LIN {X 0,Y 580.04,Z 560.279,A -85,B 0,C 180,E1 -1982.083,E2 -1982.083} C_VEL
LIN {X 0,Y 580.123,Z 557.073,A -85,B 0,C 180,E1 -1983.473,E2 -1983.473} C_VEL
LIN {X 0,Y 580.108,Z 553.521,A -85,B 0,C 180,E1 -1984.517,E2 -1984.517} C_VEL
LIN {X 0,Y 580.137,Z 548.87,A -85,B 0,C 180,E1 -1985.562,E2 -1985.562} C_VEL
LIN {X 0,Y 580.13,Z 542.972,A -85,B 0,C 180,E1 -1986.611,E2 -1986.611} C_VEL
LIN {X 0,Y 580.221,Z 535.668,A -85,B 0,C 180,E1 -1987.657,E2 -1987.657} C_VEL
LIN {X 0,Y 580.259,Z 526.563,A -85,B 0,C 180,E1 -1988.708,E2 -1988.708} C_VEL
LIN {X 0,Y 580.369,Z 515.986,A -85,B 0,C 180,E1 -1989.673,E2 -1989.673} C_VEL
LIN {X 0,Y 580.453,Z 506.507,A -85,B 0,C 180,E1 -1990.376,E2 -1990.376} C_VEL
LIN {X 0,Y 580.558,Z 496.346,A -85,B 0,C 180,E1 -1990.992,E2 -1990.992} C_VEL
LIN {X 0,Y 580.6,Z 486.208,A -85,B 0,C 180,E1 -1991.486,E2 -1991.486} C_VEL
LIN {X 0,Y 580.71,Z 474.792,A -85,B 0,C 180,E1 -1991.917,E2 -1991.917} C_VEL
LIN {X 0,Y 580.801,Z 461.468,A -85,B 0,C 180,E1 -1992.27,E2 -1992.27} C_VEL
LIN {X 0,Y 580.831,Z 443.197,A -85,B 0,C 180,E1 -1992.535,E2 -1992.535} C_VEL
LIN {X 0,Y 580.93,Z 408.349,A -85,B 0,C 180,E1 -1992.966,E2 -1992.966} C_VEL
LIN {X 0,Y 580.085,Z 398.577,A -85,B 0,C 180,E1 -1993.118,E2 -1993.118} C_VEL
LIN {X 0,Y 578.705,Z 392.854,A -85,B 0,C 180,E1 -1993.21,E2 -1993.21} C_VEL
LIN {X 0,Y 574.137,Z 379.962,A -85,B 0,C 180,E1 -1993.479,E2 -1993.479} C_VEL
LIN {X 0,Y 573.484,Z 378.185,A -85,B 0,C 180,E1 -1993.53,E2 -1993.53} C_VEL
LIN {X 0,Y 573.292,Z 377.197,A -85,B 0,C 180,E1 -1993.65,E2 -1993.65} C_VEL
LIN {X 0,Y 573.25,Z 377.078,A -85,B 0,C 180,E1 -1996.378,E2 -1996.378} C_VEL
LIN {X 0,Y 573.27,Z 377.074,A -85,B 0,C 180,E1 -1999.33,E2 -1999.33} C_VEL
LIN {X 0,Y 573.237,Z 377.078,A -85,B 0,C 180,E1 -2002.338,E2 -2002.338} C_VEL
LIN {X 0,Y 573.248,Z 377.074,A -85,B 0,C 180,E1 -2005.411,E2 -2005.411} C_VEL
LIN {X 0,Y 573.232,Z 377.081,A -85,B 0,C 180,E1 -2008.565,E2 -2008.565} C_VEL
LIN {X 0,Y 573.227,Z 377.082,A -85,B 0,C 180,E1 -2010.993,E2 -2010.993} C_VEL
LIN {X 0,Y 573.244,Z 377.072,A -85,B 0,C 180,E1 -2013.521,E2 -2013.521} C_VEL
LIN {X 0,Y 573.197,Z 377.081,A -85,B 0,C 180,E1 -2016.053,E2 -2016.053} C_VEL
LIN {X 0,Y 573.242,Z 377.083,A -85,B 0,C 180,E1 -2018.702,E2 -2018.702} C_VEL
LIN {X 0,Y 573.23,Z 377.075,A -85,B 0,C 180,E1 -2021.593,E2 -2021.593} C_VEL
LIN {X 0,Y 573.22,Z 377.082,A -85,B 0,C 180,E1 -2024.335,E2 -2024.335} C_VEL
LIN {X 0,Y 573.236,Z 377.075,A -85,B 0,C 180,E1 -2027.359,E2 -2027.359} C_VEL
LIN {X 0,Y 573.239,Z 377.082,A -85,B 0,C 180,E1 -2030.392,E2 -2030.392} C_VEL
LIN {X 0,Y 573.233,Z 377.078,A -85,B 0,C 180,E1 -2033.076,E2 -2033.076} C_VEL
LIN {X 0,Y 573.265,Z 377.071,A -85,B 0,C 180,E1 -2035.671,E2 -2035.671} C_VEL
LIN {X 0,Y 573.238,Z 377.078,A -85,B 0,C 180,E1 -2038.184,E2 -2038.184} C_VEL
LIN {X 0,Y 573.258,Z 377.081,A -85,B 0,C 180,E1 -2040.634,E2 -2040.634} C_VEL
LIN {X 0,Y 573.297,Z 377.287,A -85,B 0,C 180,E1 -2043.388,E2 -2043.388} C_VEL
LIN {X 0,Y 574.525,Z 382.647,A -85,B 0,C 180,E1 -2044.067,E2 -2044.067} C_VEL
LIN {X 0,Y 574.55,Z 397.786,A -85,B 0,C 180,E1 -2045.809,E2 -2045.809} C_VEL
LIN {X 0,Y 574.254,Z 421.464,A -85,B 0,C 180,E1 -2048.586,E2 -2048.586} C_VEL
LIN {X 0,Y 573.914,Z 446.146,A -85,B 0,C 180,E1 -2051.434,E2 -2051.434} C_VEL
LIN {X 0,Y 573.616,Z 471.912,A -85,B 0,C 180,E1 -2054.363,E2 -2054.363} C_VEL
LIN {X 0,Y 573.514,Z 488.192,A -85,B 0,C 180,E1 -2056.175,E2 -2056.175} C_VEL
LIN {X 0,Y 574.082,Z 493.73,A -85,B 0,C 180,E1 -2056.279,E2 -2056.279} C_VEL
LIN {X 0,Y 573.886,Z 597.916,A -85,B 0,C 180,E1 -2057.602,E2 -2057.602} C_VEL
LIN {X 0,Y 573.831,Z 610.341,A -85,B 0,C 180,E1 -2057.893,E2 -2057.893} C_VEL
LIN {X 0,Y 573.705,Z 622.21,A -85,B 0,C 180,E1 -2058.294,E2 -2058.294} C_VEL
LIN {X 0,Y 573.588,Z 634.849,A -85,B 0,C 180,E1 -2058.876,E2 -2058.876} C_VEL
LIN {X 0,Y 573.445,Z 646.523,A -85,B 0,C 180,E1 -2059.585,E2 -2059.585} C_VEL
LIN {X 0,Y 573.35,Z 655.955,A -85,B 0,C 180,E1 -2060.297,E2 -2060.297} C_VEL
LIN {X 0,Y 573.262,Z 663.842,A -85,B 0,C 180,E1 -2061.007,E2 -2061.007} C_VEL
LIN {X 0,Y 573.178,Z 672.073,A -85,B 0,C 180,E1 -2061.894,E2 -2061.894} C_VEL
LIN {X 0,Y 573.105,Z 680.149,A -85,B 0,C 180,E1 -2062.956,E2 -2062.956} C_VEL
LIN {X 0,Y 573.093,Z 686.626,A -85,B 0,C 180,E1 -2064.017,E2 -2064.017} C_VEL
LIN {X 0,Y 572.962,Z 691.755,A -85,B 0,C 180,E1 -2065.074,E2 -2065.074} C_VEL
LIN {X 0,Y 573.014,Z 695.735,A -85,B 0,C 180,E1 -2066.132,E2 -2066.132} C_VEL
LIN {X 0,Y 572.959,Z 698.688,A -85,B 0,C 180,E1 -2067.188,E2 -2067.188} C_VEL
LIN {X 0,Y 572.939,Z 700.137,A -85,B 0,C 180,E1 -2067.891,E2 -2067.891} C_VEL
LIN {X 0,Y 572.941,Z 701.756,A -85,B 0,C 180,E1 -2069.297,E2 -2069.297} C_VEL
LIN {X 0,Y 572.939,Z 701.996,A -85,B 0,C 180,E1 -2070,E2 -2070} C_VEL
LIN {X 0,Y 572.947,Z 701.229,A -85,B 0,C 180,E1 -2071.406,E2 -2071.406} C_VEL
LIN {X 0,Y 572.939,Z 700.28,A -85,B 0,C 180,E1 -2072.109,E2 -2072.109} C_VEL
LIN {X 0,Y 572.959,Z 698.879,A -85,B 0,C 180,E1 -2072.812,E2 -2072.812} C_VEL
LIN {X 0,Y 573.015,Z 696.005,A -85,B 0,C 180,E1 -2073.868,E2 -2073.868} C_VEL
LIN {X 0,Y 572.962,Z 692.116,A -85,B 0,C 180,E1 -2074.926,E2 -2074.926} C_VEL
LIN {X 0,Y 573.071,Z 687.095,A -85,B 0,C 180,E1 -2075.984,E2 -2075.984} C_VEL
LIN {X 0,Y 573.114,Z 679.539,A -85,B 0,C 180,E1 -2077.221,E2 -2077.221} C_VEL
LIN {X 0,Y 573.169,Z 672.832,A -85,B 0,C 180,E1 -2078.106,E2 -2078.106} C_VEL
LIN {X 0,Y 573.251,Z 664.745,A -85,B 0,C 180,E1 -2078.993,E2 -2078.993} C_VEL
LIN {X 0,Y 573.342,Z 654.904,A -85,B 0,C 180,E1 -2079.882,E2 -2079.882} C_VEL
LIN {X 0,Y 573.516,Z 643.899,A -85,B 0,C 180,E1 -2080.681,E2 -2080.681} C_VEL
LIN {X 0,Y 573.636,Z 631.59,A -85,B 0,C 180,E1 -2081.377,E2 -2081.377} C_VEL
LIN {X 0,Y 573.701,Z 620.22,A -85,B 0,C 180,E1 -2081.872,E2 -2081.872} C_VEL
LIN {X 0,Y 573.802,Z 608.017,A -85,B 0,C 180,E1 -2082.265,E2 -2082.265} C_VEL
LIN {X 0,Y 573.922,Z 595.156,A -85,B 0,C 180,E1 -2082.532,E2 -2082.532} C_VEL
LIN {X 0,Y 573.944,Z 491.455,A -85,B 0,C 180,E1 -2083.843,E2 -2083.843} C_VEL
LIN {X 0,Y 573.528,Z 488.15,A -85,B 0,C 180,E1 -2083.915,E2 -2083.915} C_VEL
LIN {X 0,Y 573.733,Z 461.428,A -85,B 0,C 180,E1 -2086.914,E2 -2086.914} C_VEL
LIN {X 0,Y 574.055,Z 435.714,A -85,B 0,C 180,E1 -2089.853,E2 -2089.853} C_VEL
LIN {X 0,Y 574.423,Z 409.87,A -85,B 0,C 180,E1 -2092.859,E2 -2092.859} C_VEL
LIN {X 0,Y 574.656,Z 388.489,A -85,B 0,C 180,E1 -2095.344,E2 -2095.344} C_VEL
LIN {X 0,Y 574.626,Z 383.426,A -85,B 0,C 180,E1 -2095.928,E2 -2095.928} C_VEL
LIN {X 0,Y 573.246,Z 377.157,A -85,B 0,C 180,E1 -2096.74,E2 -2096.74} C_VEL
LIN {X 0,Y 573.226,Z 377.079,A -85,B 0,C 180,E1 -2099.484,E2 -2099.484} C_VEL
LIN {X 0,Y 573.24,Z 377.077,A -85,B 0,C 180,E1 -2102.226,E2 -2102.226} C_VEL
LIN {X 0,Y 573.225,Z 377.077,A -85,B 0,C 180,E1 -2104.769,E2 -2104.769} C_VEL
LIN {X 0,Y 573.223,Z 377.084,A -85,B 0,C 180,E1 -2107.809,E2 -2107.809} C_VEL
LIN {X 0,Y 573.249,Z 377.071,A -85,B 0,C 180,E1 -2110.525,E2 -2110.525} C_VEL
LIN {X 0,Y 573.207,Z 377.086,A -85,B 0,C 180,E1 -2113.665,E2 -2113.665} C_VEL
LIN {X 0,Y 573.204,Z 377.078,A -85,B 0,C 180,E1 -2116.637,E2 -2116.637} C_VEL
LIN {X 0,Y 573.249,Z 377.08,A -85,B 0,C 180,E1 -2119.475,E2 -2119.475} C_VEL
LIN {X 0,Y 573.221,Z 377.078,A -85,B 0,C 180,E1 -2122.191,E2 -2122.191} C_VEL
LIN {X 0,Y 573.222,Z 377.079,A -85,B 0,C 180,E1 -2125.231,E2 -2125.231} C_VEL
LIN {X 0,Y 573.252,Z 377.082,A -85,B 0,C 180,E1 -2127.773,E2 -2127.773} C_VEL
LIN {X 0,Y 573.225,Z 377.075,A -85,B 0,C 180,E1 -2130.632,E2 -2130.632} C_VEL
LIN {X 0,Y 573.201,Z 377.086,A -85,B 0,C 180,E1 -2133.516,E2 -2133.516} C_VEL
LIN {X 0,Y 573.219,Z 377.078,A -85,B 0,C 180,E1 -2136.134,E2 -2136.134} C_VEL
LIN {X 0,Y 573.234,Z 377.077,A -85,B 0,C 180,E1 -2139.173,E2 -2139.173} C_VEL
LIN {X 0,Y 573.202,Z 377.083,A -85,B 0,C 180,E1 -2141.41,E2 -2141.41} C_VEL
LIN {X 0,Y 573.211,Z 377.079,A -85,B 0,C 180,E1 -2144.351,E2 -2144.351} C_VEL
LIN {X 0,Y 573.214,Z 377.077,A -85,B 0,C 180,E1 -2146.529,E2 -2146.529} C_VEL
LIN {X 0,Y 573.242,Z 377.075,A -85,B 0,C 180,E1 -2149.403,E2 -2149.403} C_VEL
LIN {X 0,Y 573.223,Z 377.078,A -85,B 0,C 180,E1 -2152.249,E2 -2152.249} C_VEL
LIN {X 0,Y 573.281,Z 377.067,A -85,B 0,C 180,E1 -2155.077,E2 -2155.077} C_VEL
LIN {X 0,Y 573.309,Z 377.073,A -85,B 0,C 180,E1 -2157.892,E2 -2157.892} C_VEL
LIN {X 0,Y 573.32,Z 377.069,A -85,B 0,C 180,E1 -2160,E2 -2160} C_VEL
LIN {X 0,Y 573.273,Z 377.066,A -85,B 0,C 180,E1 -2162.811,E2 -2162.811} C_VEL
LIN {X 0,Y 573.27,Z 377.077,A -85,B 0,C 180,E1 -2165.628,E2 -2165.628} C_VEL
LIN {X 0,Y 573.238,Z 377.073,A -85,B 0,C 180,E1 -2168.46,E2 -2168.46} C_VEL
LIN {X 0,Y 573.24,Z 377.075,A -85,B 0,C 180,E1 -2171.313,E2 -2171.313} C_VEL
LIN {X 0,Y 573.246,Z 377.074,A -85,B 0,C 180,E1 -2174.408,E2 -2174.408} C_VEL
LIN {X 0,Y 573.18,Z 377.079,A -85,B 0,C 180,E1 -2177.114,E2 -2177.114} C_VEL
LIN {X 0,Y 573.204,Z 377.084,A -85,B 0,C 180,E1 -2180.078,E2 -2180.078} C_VEL
LIN {X 0,Y 573.218,Z 377.077,A -85,B 0,C 180,E1 -2182.339,E2 -2182.339} C_VEL
LIN {X 0,Y 573.209,Z 377.081,A -85,B 0,C 180,E1 -2185.412,E2 -2185.412} C_VEL
LIN {X 0,Y 573.195,Z 377.084,A -85,B 0,C 180,E1 -2188.017,E2 -2188.017} C_VEL
LIN {X 0,Y 573.22,Z 377.076,A -85,B 0,C 180,E1 -2190.88,E2 -2190.88} C_VEL
LIN {X 0,Y 573.245,Z 377.078,A -85,B 0,C 180,E1 -2193.521,E2 -2193.521} C_VEL
LIN {X 0,Y 573.184,Z 377.088,A -85,B 0,C 180,E1 -2196.054,E2 -2196.054} C_VEL
LIN {X 0,Y 573.215,Z 377.076,A -85,B 0,C 180,E1 -2198.704,E2 -2198.704} C_VEL
LIN {X 0,Y 573.187,Z 377.08,A -85,B 0,C 180,E1 -2201.587,E2 -2201.587} C_VEL
LIN {X 0,Y 573.207,Z 377.081,A -85,B 0,C 180,E1 -2204.336,E2 -2204.336} C_VEL
LIN {X 0,Y 573.195,Z 377.079,A -85,B 0,C 180,E1 -2206.636,E2 -2206.636} C_VEL
LIN {X 0,Y 573.202,Z 377.077,A -85,B 0,C 180,E1 -2209.48,E2 -2209.48} C_VEL
LIN {X 0,Y 573.209,Z 377.084,A -85,B 0,C 180,E1 -2212.19,E2 -2212.19} C_VEL
LIN {X 0,Y 573.211,Z 377.079,A -85,B 0,C 180,E1 -2215.233,E2 -2215.233} C_VEL
LIN {X 0,Y 573.223,Z 377.085,A -85,B 0,C 180,E1 -2217.777,E2 -2217.777} C_VEL
LIN {X 0,Y 573.219,Z 377.081,A -85,B 0,C 180,E1 -2220.631,E2 -2220.631} C_VEL
LIN {X 0,Y 573.226,Z 377.225,A -85,B 0,C 180,E1 -2222.751,E2 -2222.751} C_VEL
LIN {X 0,Y 574.782,Z 383.948,A -85,B 0,C 180,E1 -2223.589,E2 -2223.589} C_VEL
LIN {X 0,Y 574.627,Z 405.704,A -85,B 0,C 180,E1 -2226.004,E2 -2226.004} C_VEL
LIN {X 0,Y 574.261,Z 431.045,A -85,B 0,C 180,E1 -2228.85,E2 -2228.85} C_VEL
LIN {X 0,Y 573.894,Z 457.816,A -85,B 0,C 180,E1 -2231.803,E2 -2231.803} C_VEL
LIN {X 0,Y 573.643,Z 483.031,A -85,B 0,C 180,E1 -2234.545,E2 -2234.545} C_VEL
LIN {X 0,Y 573.519,Z 497.889,A -85,B 0,C 180,E1 -2236.13,E2 -2236.13} C_VEL
LIN {X 0,Y 574.08,Z 503.704,A -85,B 0,C 180,E1 -2236.234,E2 -2236.234} C_VEL
LIN {X 0,Y 573.882,Z 607.937,A -85,B 0,C 180,E1 -2237.557,E2 -2237.557} C_VEL
LIN {X 0,Y 573.785,Z 621.213,A -85,B 0,C 180,E1 -2237.869,E2 -2237.869} C_VEL
LIN {X 0,Y 573.702,Z 634.147,A -85,B 0,C 180,E1 -2238.325,E2 -2238.325} C_VEL
LIN {X 0,Y 573.591,Z 645.717,A -85,B 0,C 180,E1 -2238.878,E2 -2238.878} C_VEL
LIN {X 0,Y 573.438,Z 657.2,A -85,B 0,C 180,E1 -2239.585,E2 -2239.585} C_VEL
LIN {X 0,Y 573.331,Z 667.598,A -85,B 0,C 180,E1 -2240.385,E2 -2240.385} C_VEL
LIN {X 0,Y 573.241,Z 676.111,A -85,B 0,C 180,E1 -2241.184,E2 -2241.184} C_VEL
LIN {X 0,Y 573.161,Z 683.959,A -85,B 0,C 180,E1 -2242.071,E2 -2242.071} C_VEL
LIN {X 0,Y 573.073,Z 691.953,A -85,B 0,C 180,E1 -2243.185,E2 -2243.185} C_VEL
LIN {X 0,Y 573.07,Z 698.679,A -85,B 0,C 180,E1 -2244.37,E2 -2244.37} C_VEL
LIN {X 0,Y 573.028,Z 703.371,A -85,B 0,C 180,E1 -2245.427,E2 -2245.427} C_VEL
LIN {X 0,Y 573.022,Z 706.957,A -85,B 0,C 180,E1 -2246.484,E2 -2246.484} C_VEL
LIN {X 0,Y 572.959,Z 708.808,A -85,B 0,C 180,E1 -2247.188,E2 -2247.188} C_VEL
LIN {X 0,Y 572.939,Z 710.198,A -85,B 0,C 180,E1 -2247.891,E2 -2247.891} C_VEL
LIN {X 0,Y 572.94,Z 711.785,A -85,B 0,C 180,E1 -2249.297,E2 -2249.297} C_VEL
LIN {X 0,Y 572.938,Z 712,A -85,B 0,C 180,E1 -2250,E2 -2250} C_VEL
LIN {X 0,Y 572.946,Z 711.186,A -85,B 0,C 180,E1 -2251.406,E2 -2251.406} C_VEL
LIN {X 0,Y 572.939,Z 710.2,A -85,B 0,C 180,E1 -2252.109,E2 -2252.109} C_VEL
LIN {X 0,Y 572.959,Z 708.81,A -85,B 0,C 180,E1 -2252.812,E2 -2252.812} C_VEL
LIN {X 0,Y 573.015,Z 705.896,A -85,B 0,C 180,E1 -2253.868,E2 -2253.868} C_VEL
LIN {X 0,Y 572.963,Z 701.949,A -85,B 0,C 180,E1 -2254.926,E2 -2254.926} C_VEL
LIN {X 0,Y 573.064,Z 695.877,A -85,B 0,C 180,E1 -2256.16,E2 -2256.16} C_VEL
LIN {X 0,Y 573.119,Z 689.238,A -85,B 0,C 180,E1 -2257.221,E2 -2257.221} C_VEL
LIN {X 0,Y 573.201,Z 680.991,A -85,B 0,C 180,E1 -2258.283,E2 -2258.283} C_VEL
LIN {X 0,Y 573.287,Z 672.539,A -85,B 0,C 180,E1 -2259.17,E2 -2259.17} C_VEL
LIN {X 0,Y 573.425,Z 662.098,A -85,B 0,C 180,E1 -2260.058,E2 -2260.058} C_VEL
LIN {X 0,Y 573.534,Z 651.772,A -85,B 0,C 180,E1 -2260.769,E2 -2260.769} C_VEL
LIN {X 0,Y 573.628,Z 640.588,A -85,B 0,C 180,E1 -2261.385,E2 -2261.385} C_VEL
LIN {X 0,Y 573.719,Z 628.768,A -85,B 0,C 180,E1 -2261.885,E2 -2261.885} C_VEL
LIN {X 0,Y 573.822,Z 615.349,A -85,B 0,C 180,E1 -2262.287,E2 -2262.287} C_VEL
LIN {X 0,Y 573.951,Z 602.085,A -85,B 0,C 180,E1 -2262.531,E2 -2262.531} C_VEL
LIN {X 0,Y 573.89,Z 500.813,A -85,B 0,C 180,E1 -2263.807,E2 -2263.807} C_VEL
LIN {X 0,Y 573.519,Z 497.888,A -85,B 0,C 180,E1 -2263.87,E2 -2263.87} C_VEL
LIN {X 0,Y 573.782,Z 472.947,A -85,B 0,C 180,E1 -2266.546,E2 -2266.546} C_VEL
LIN {X 0,Y 574.04,Z 446.069,A -85,B 0,C 180,E1 -2269.487,E2 -2269.487} C_VEL
LIN {X 0,Y 574.394,Z 420.835,A -85,B 0,C 180,E1 -2272.29,E2 -2272.29} C_VEL
LIN {X 0,Y 574.659,Z 399.163,A -85,B 0,C 180,E1 -2274.721,E2 -2274.721} C_VEL
LIN {X 0,Y 574.682,Z 383.397,A -85,B 0,C 180,E1 -2276.416,E2 -2276.416} C_VEL
LIN {X 0,Y 573.222,Z 377.203,A -85,B 0,C 180,E1 -2277.175,E2 -2277.175} C_VEL
LIN {X 0,Y 573.218,Z 377.086,A -85,B 0,C 180,E1 -2280.178,E2 -2280.178} C_VEL
LIN {X 0,Y 573.217,Z 377.079,A -85,B 0,C 180,E1 -2282.647,E2 -2282.647} C_VEL
LIN {X 0,Y 573.18,Z 377.084,A -85,B 0,C 180,E1 -2285.19,E2 -2285.19} C_VEL
LIN {X 0,Y 573.211,Z 377.087,A -85,B 0,C 180,E1 -2287.81,E2 -2287.81} C_VEL
LIN {X 0,Y 573.201,Z 377.08,A -85,B 0,C 180,E1 -2290.529,E2 -2290.529} C_VEL
LIN {X 0,Y 573.196,Z 377.084,A -85,B 0,C 180,E1 -2293.363,E2 -2293.363} C_VEL
LIN {X 0,Y 573.206,Z 377.08,A -85,B 0,C 180,E1 -2296.335,E2 -2296.335} C_VEL
LIN {X 0,Y 573.204,Z 377.079,A -85,B 0,C 180,E1 -2298.54,E2 -2298.54} C_VEL
LIN {X 0,Y 573.233,Z 377.08,A -85,B 0,C 180,E1 -2301.297,E2 -2301.297} C_VEL
LIN {X 0,Y 573.188,Z 377.085,A -85,B 0,C 180,E1 -2304.022,E2 -2304.022} C_VEL
LIN {X 0,Y 573.242,Z 377.075,A -85,B 0,C 180,E1 -2306.516,E2 -2306.516} C_VEL
LIN {X 0,Y 573.228,Z 377.08,A -85,B 0,C 180,E1 -2309.119,E2 -2309.119} C_VEL
LIN {X 0,Y 573.228,Z 377.085,A -85,B 0,C 180,E1 -2311.435,E2 -2311.435} C_VEL
LIN {X 0,Y 573.24,Z 377.075,A -85,B 0,C 180,E1 -2314.589,E2 -2314.589} C_VEL
LIN {X 0,Y 573.235,Z 377.081,A -85,B 0,C 180,E1 -2317.662,E2 -2317.662} C_VEL
LIN {X 0,Y 573.269,Z 377.073,A -85,B 0,C 180,E1 -2320.67,E2 -2320.67} C_VEL
LIN {X 0,Y 573.251,Z 377.08,A -85,B 0,C 180,E1 -2323.622,E2 -2323.622} C_VEL
LIN {X 0,Y 573.299,Z 377.197,A -85,B 0,C 180,E1 -2326.441,E2 -2326.441} C_VEL
LIN {X 0,Y 573.526,Z 378.312,A -85,B 0,C 180,E1 -2326.567,E2 -2326.567} C_VEL
LIN {X 0,Y 574.033,Z 380.55,A -85,B 0,C 180,E1 -2326.616,E2 -2326.616} C_VEL
LIN {X 0,Y 573.912,Z 457.586,A -85,B 0,C 180,E1 -2327.603,E2 -2327.603} C_VEL
LIN {X 0,Y 573.807,Z 468.697,A -85,B 0,C 180,E1 -2327.848,E2 -2327.848} C_VEL
LIN {X 0,Y 573.718,Z 481.135,A -85,B 0,C 180,E1 -2328.249,E2 -2328.249} C_VEL
LIN {X 0,Y 573.622,Z 493.628,A -85,B 0,C 180,E1 -2328.813,E2 -2328.813} C_VEL
LIN {X 0,Y 573.488,Z 503.829,A -85,B 0,C 180,E1 -2329.408,E2 -2329.408} C_VEL
LIN {X 0,Y 573.343,Z 513.737,A -85,B 0,C 180,E1 -2330.118,E2 -2330.118} C_VEL
LIN {X 0,Y 573.287,Z 521.975,A -85,B 0,C 180,E1 -2330.83,E2 -2330.83} C_VEL
LIN {X 0,Y 573.187,Z 530.527,A -85,B 0,C 180,E1 -2331.717,E2 -2331.717} C_VEL
LIN {X 0,Y 573.114,Z 537.611,A -85,B 0,C 180,E1 -2332.602,E2 -2332.602} C_VEL
LIN {X 0,Y 573.049,Z 544.597,A -85,B 0,C 180,E1 -2333.663,E2 -2333.663} C_VEL
LIN {X 0,Y 573.009,Z 550.176,A -85,B 0,C 180,E1 -2334.722,E2 -2334.722} C_VEL
LIN {X 0,Y 573.031,Z 554.536,A -85,B 0,C 180,E1 -2335.78,E2 -2335.78} C_VEL
LIN {X 0,Y 572.959,Z 558.66,A -85,B 0,C 180,E1 -2337.188,E2 -2337.188} C_VEL
LIN {X 0,Y 572.939,Z 560.134,A -85,B 0,C 180,E1 -2337.891,E2 -2337.891} C_VEL
LIN {X 0,Y 572.941,Z 561.735,A -85,B 0,C 180,E1 -2339.297,E2 -2339.297} C_VEL
LIN {X 0,Y 572.939,Z 561.996,A -85,B 0,C 180,E1 -2340,E2 -2340} C_VEL
LIN {X 0,Y 572.947,Z 561.225,A -85,B 0,C 180,E1 -2341.406,E2 -2341.406} C_VEL
LIN {X 0,Y 572.939,Z 560.28,A -85,B 0,C 180,E1 -2342.109,E2 -2342.109} C_VEL
LIN {X 0,Y 573.022,Z 557.067,A -85,B 0,C 180,E1 -2343.516,E2 -2343.516} C_VEL
LIN {X 0,Y 573.028,Z 553.51,A -85,B 0,C 180,E1 -2344.573,E2 -2344.573} C_VEL
LIN {X 0,Y 573.068,Z 548.857,A -85,B 0,C 180,E1 -2345.63,E2 -2345.63} C_VEL
LIN {X 0,Y 573.051,Z 543.428,A -85,B 0,C 180,E1 -2346.617,E2 -2346.617} C_VEL
LIN {X 0,Y 573.142,Z 536.965,A -85,B 0,C 180,E1 -2347.575,E2 -2347.575} C_VEL
LIN {X 0,Y 573.216,Z 529.755,A -85,B 0,C 180,E1 -2348.461,E2 -2348.461} C_VEL
LIN {X 0,Y 573.286,Z 522.915,A -85,B 0,C 180,E1 -2349.17,E2 -2349.17} C_VEL
LIN {X 0,Y 573.335,Z 514.855,A -85,B 0,C 180,E1 -2349.882,E2 -2349.882} C_VEL
LIN {X 0,Y 573.454,Z 506.478,A -85,B 0,C 180,E1 -2350.504,E2 -2350.504} C_VEL
LIN {X 0,Y 573.56,Z 497.918,A -85,B 0,C 180,E1 -2351.038,E2 -2351.038} C_VEL
LIN {X 0,Y 573.636,Z 487.583,A -85,B 0,C 180,E1 -2351.564,E2 -2351.564} C_VEL
LIN {X 0,Y 573.735,Z 477.316,A -85,B 0,C 180,E1 -2351.975,E2 -2351.975} C_VEL
LIN {X 0,Y 573.829,Z 466.957,A -85,B 0,C 180,E1 -2352.287,E2 -2352.287} C_VEL
LIN {X 0,Y 573.935,Z 456.287,A -85,B 0,C 180,E1 -2352.509,E2 -2352.509} C_VEL
LIN {X 0,Y 573.892,Z 379.538,A -85,B 0,C 180,E1 -2353.49,E2 -2353.49} C_VEL
LIN {X 0,Y 573.484,Z 378.185,A -85,B 0,C 180,E1 -2353.53,E2 -2353.53} C_VEL
LIN {X 0,Y 572.836,Z 377.298,A -85,B 0,C 180,E1 -2353.661,E2 -2353.661} C_VEL
LIN {X 0,Y 569.914,Z 377.495,A -85,B 0,C 180,E1 -2354.45,E2 -2354.45} C_VEL
LIN {X 0,Y 567.817,Z 378.138,A -85,B 0,C 180,E1 -2355.262,E2 -2355.262} C_VEL
LIN {X 0,Y 566.425,Z 378.06,A -85,B 0,C 180,E1 -2356.16,E2 -2356.16} C_VEL
LIN {X 0,Y 566.216,Z 377.957,A -85,B 0,C 180,E1 -2356.616,E2 -2356.616} C_VEL
LIN {X 0,Y 566.206,Z 377.952,A -85,B 0,C 180,E1 -2359.581,E2 -2359.581} C_VEL
LIN {X 0,Y 566.196,Z 377.952,A -85,B 0,C 180,E1 -2361.863,E2 -2361.863} C_VEL
LIN {X 0,Y 566.222,Z 377.954,A -85,B 0,C 180,E1 -2365.03,E2 -2365.03} C_VEL
LIN {X 0,Y 566.178,Z 377.954,A -85,B 0,C 180,E1 -2367.341,E2 -2367.341} C_VEL
LIN {X 0,Y 566.204,Z 377.949,A -85,B 0,C 180,E1 -2369.769,E2 -2369.769} C_VEL
LIN {X 0,Y 566.206,Z 377.956,A -85,B 0,C 180,E1 -2372.43,E2 -2372.43} C_VEL
LIN {X 0,Y 566.183,Z 377.959,A -85,B 0,C 180,E1 -2374.989,E2 -2374.989} C_VEL
LIN {X 0,Y 566.195,Z 377.951,A -85,B 0,C 180,E1 -2377.461,E2 -2377.461} C_VEL
LIN {X 0,Y 566.209,Z 377.953,A -85,B 0,C 180,E1 -2380.199,E2 -2380.199} C_VEL
LIN {X 0,Y 566.19,Z 377.956,A -85,B 0,C 180,E1 -2383.056,E2 -2383.056} C_VEL
LIN {X 0,Y 566.195,Z 377.953,A -85,B 0,C 180,E1 -2386.049,E2 -2386.049} C_VEL
LIN {X 0,Y 566.206,Z 377.952,A -85,B 0,C 180,E1 -2389.215,E2 -2389.215} C_VEL
LIN {X 0,Y 566.183,Z 377.95,A -85,B 0,C 180,E1 -2391.636,E2 -2391.636} C_VEL
LIN {X 0,Y 566.152,Z 377.964,A -85,B 0,C 180,E1 -2394.307,E2 -2394.307} C_VEL
LIN {X 0,Y 566.222,Z 377.952,A -85,B 0,C 180,E1 -2396.898,E2 -2396.898} C_VEL
LIN {X 0,Y 566.174,Z 377.955,A -85,B 0,C 180,E1 -2399.407,E2 -2399.407} C_VEL
LIN {X 0,Y 566.19,Z 377.956,A -85,B 0,C 180,E1 -2401.856,E2 -2401.856} C_VEL
LIN {X 0,Y 566.24,Z 378.094,A -85,B 0,C 180,E1 -2403.199,E2 -2403.199} C_VEL
LIN {X 0,Y 567.724,Z 385.361,A -85,B 0,C 180,E1 -2404.128,E2 -2404.128} C_VEL
LIN {X 0,Y 567.562,Z 408.907,A -85,B 0,C 180,E1 -2406.849,E2 -2406.849} C_VEL
LIN {X 0,Y 567.23,Z 433.269,A -85,B 0,C 180,E1 -2409.701,E2 -2409.701} C_VEL
LIN {X 0,Y 566.818,Z 457.423,A -85,B 0,C 180,E1 -2412.502,E2 -2412.502} C_VEL
LIN {X 0,Y 566.609,Z 482.281,A -85,B 0,C 180,E1 -2415.349,E2 -2415.349} C_VEL
LIN {X 0,Y 566.551,Z 488.21,A -85,B 0,C 180,E1 -2416.002,E2 -2416.002} C_VEL
LIN {X 0,Y 567.198,Z 493.776,A -85,B 0,C 180,E1 -2416.109,E2 -2416.109} C_VEL
LIN {X 0,Y 566.976,Z 597.941,A -85,B 0,C 180,E1 -2417.449,E2 -2417.449} C_VEL
LIN {X 0,Y 566.912,Z 610.337,A -85,B 0,C 180,E1 -2417.743,E2 -2417.743} C_VEL
LIN {X 0,Y 566.743,Z 621.034,A -85,B 0,C 180,E1 -2418.103,E2 -2418.103} C_VEL
LIN {X 0,Y 566.661,Z 631.226,A -85,B 0,C 180,E1 -2418.554,E2 -2418.554} C_VEL
LIN {X 0,Y 566.561,Z 642.595,A -85,B 0,C 180,E1 -2419.193,E2 -2419.193} C_VEL
LIN {X 0,Y 566.35,Z 653.833,A -85,B 0,C 180,E1 -2419.995,E2 -2419.995} C_VEL
LIN {X 0,Y 566.234,Z 663.839,A -85,B 0,C 180,E1 -2420.895,E2 -2420.895} C_VEL
LIN {X 0,Y 566.133,Z 672.069,A -85,B 0,C 180,E1 -2421.792,E2 -2421.792} C_VEL
LIN {X 0,Y 566.041,Z 680.151,A -85,B 0,C 180,E1 -2422.868,E2 -2422.868} C_VEL
LIN {X 0,Y 566.003,Z 686.629,A -85,B 0,C 180,E1 -2423.942,E2 -2423.942} C_VEL
LIN {X 0,Y 565.877,Z 691.754,A -85,B 0,C 180,E1 -2425.013,E2 -2425.013} C_VEL
LIN {X 0,Y 565.926,Z 695.732,A -85,B 0,C 180,E1 -2426.084,E2 -2426.084} C_VEL
LIN {X 0,Y 565.877,Z 698.683,A -85,B 0,C 180,E1 -2427.153,E2 -2427.153} C_VEL
LIN {X 0,Y 565.84,Z 700.138,A -85,B 0,C 180,E1 -2427.865,E2 -2427.865} C_VEL
LIN {X 0,Y 565.841,Z 701.751,A -85,B 0,C 180,E1 -2429.288,E2 -2429.288} C_VEL
LIN {X 0,Y 565.839,Z 701.996,A -85,B 0,C 180,E1 -2430,E2 -2430} C_VEL
LIN {X 0,Y 565.846,Z 701.228,A -85,B 0,C 180,E1 -2431.424,E2 -2431.424} C_VEL
LIN {X 0,Y 565.84,Z 700.281,A -85,B 0,C 180,E1 -2432.136,E2 -2432.136} C_VEL
LIN {X 0,Y 565.878,Z 698.871,A -85,B 0,C 180,E1 -2432.848,E2 -2432.848} C_VEL
LIN {X 0,Y 565.959,Z 694.846,A -85,B 0,C 180,E1 -2434.273,E2 -2434.273} C_VEL
LIN {X 0,Y 565.937,Z 690.579,A -85,B 0,C 180,E1 -2435.344,E2 -2435.344} C_VEL
LIN {X 0,Y 565.966,Z 685.119,A -85,B 0,C 180,E1 -2436.417,E2 -2436.417} C_VEL
LIN {X 0,Y 566.054,Z 678.267,A -85,B 0,C 180,E1 -2437.491,E2 -2437.491} C_VEL
LIN {X 0,Y 566.133,Z 671.313,A -85,B 0,C 180,E1 -2438.388,E2 -2438.388} C_VEL
LIN {X 0,Y 566.249,Z 662.944,A -85,B 0,C 180,E1 -2439.285,E2 -2439.285} C_VEL
LIN {X 0,Y 566.422,Z 652.692,A -85,B 0,C 180,E1 -2440.184,E2 -2440.184} C_VEL
LIN {X 0,Y 566.532,Z 641.29,A -85,B 0,C 180,E1 -2440.977,E2 -2440.977} C_VEL
LIN {X 0,Y 566.661,Z 631.223,A -85,B 0,C 180,E1 -2441.536,E2 -2441.536} C_VEL
LIN {X 0,Y 566.756,Z 620.183,A -85,B 0,C 180,E1 -2442.02,E2 -2442.02} C_VEL
LIN {X 0,Y 566.878,Z 608.749,A -85,B 0,C 180,E1 -2442.394,E2 -2442.394} C_VEL
LIN {X 0,Y 566.993,Z 596.624,A -85,B 0,C 180,E1 -2442.665,E2 -2442.665} C_VEL
LIN {X 0,Y 567.07,Z 492.083,A -85,B 0,C 180,E1 -2444.006,E2 -2444.006} C_VEL
LIN {X 0,Y 566.575,Z 488.142,A -85,B 0,C 180,E1 -2444.09,E2 -2444.09} C_VEL
LIN {X 0,Y 566.811,Z 459.888,A -85,B 0,C 180,E1 -2447.304,E2 -2447.304} C_VEL
LIN {X 0,Y 567.173,Z 435.805,A -85,B 0,C 180,E1 -2450.093,E2 -2450.093} C_VEL
LIN {X 0,Y 567.561,Z 411.358,A -85,B 0,C 180,E1 -2452.958,E2 -2452.958} C_VEL
LIN {X 0,Y 567.762,Z 386.129,A -85,B 0,C 180,E1 -2455.871,E2 -2455.871} C_VEL
LIN {X 0,Y 566.821,Z 380.933,A -85,B 0,C 180,E1 -2456.511,E2 -2456.511} C_VEL
LIN {X 0,Y 566.212,Z 378.068,A -85,B 0,C 180,E1 -2456.9,E2 -2456.9} C_VEL
LIN {X 0,Y 566.174,Z 377.96,A -85,B 0,C 180,E1 -2459.771,E2 -2459.771} C_VEL
LIN {X 0,Y 566.196,Z 377.953,A -85,B 0,C 180,E1 -2462.428,E2 -2462.428} C_VEL
LIN {X 0,Y 566.17,Z 377.957,A -85,B 0,C 180,E1 -2464.988,E2 -2464.988} C_VEL
LIN {X 0,Y 566.189,Z 377.958,A -85,B 0,C 180,E1 -2467.462,E2 -2467.462} C_VEL
LIN {X 0,Y 566.209,Z 377.95,A -85,B 0,C 180,E1 -2470.199,E2 -2470.199} C_VEL
LIN {X 0,Y 566.151,Z 377.959,A -85,B 0,C 180,E1 -2473.059,E2 -2473.059} C_VEL
LIN {X 0,Y 566.16,Z 377.96,A -85,B 0,C 180,E1 -2476.053,E2 -2476.053} C_VEL
LIN {X 0,Y 566.159,Z 377.957,A -85,B 0,C 180,E1 -2478.859,E2 -2478.859} C_VEL
LIN {X 0,Y 566.204,Z 377.957,A -85,B 0,C 180,E1 -2481.443,E2 -2481.443} C_VEL
LIN {X 0,Y 566.142,Z 377.96,A -85,B 0,C 180,E1 -2484.306,E2 -2484.306} C_VEL
LIN {X 0,Y 566.201,Z 377.949,A -85,B 0,C 180,E1 -2486.896,E2 -2486.896} C_VEL
LIN {X 0,Y 566.172,Z 377.96,A -85,B 0,C 180,E1 -2489.407,E2 -2489.407} C_VEL
LIN {X 0,Y 566.153,Z 377.964,A -85,B 0,C 180,E1 -2491.854,E2 -2491.854} C_VEL
LIN {X 0,Y 566.187,Z 377.955,A -85,B 0,C 180,E1 -2494.25,E2 -2494.25} C_VEL
LIN {X 0,Y 566.17,Z 377.952,A -85,B 0,C 180,E1 -2496.72,E2 -2496.72} C_VEL
LIN {X 0,Y 566.198,Z 377.961,A -85,B 0,C 180,E1 -2499.662,E2 -2499.662} C_VEL
LIN {X 0,Y 566.17,Z 377.959,A -85,B 0,C 180,E1 -2501.921,E2 -2501.921} C_VEL
LIN {X 0,Y 566.188,Z 377.953,A -85,B 0,C 180,E1 -2504.89,E2 -2504.89} C_VEL
LIN {X 0,Y 566.215,Z 377.954,A -85,B 0,C 180,E1 -2507.818,E2 -2507.818} C_VEL
LIN {X 0,Y 566.187,Z 377.952,A -85,B 0,C 180,E1 -2510.714,E2 -2510.714} C_VEL
LIN {X 0,Y 566.186,Z 377.96,A -85,B 0,C 180,E1 -2513.586,E2 -2513.586} C_VEL
LIN {X 0,Y 566.173,Z 377.96,A -85,B 0,C 180,E1 -2515.729,E2 -2515.729} C_VEL
LIN {X 0,Y 566.28,Z 377.95,A -85,B 0,C 180,E1 -2517.866,E2 -2517.866} C_VEL
LIN {X 0,Y 566.288,Z 377.945,A -85,B 0,C 180,E1 -2520,E2 -2520} C_VEL
LIN {X 0,Y 566.242,Z 377.942,A -85,B 0,C 180,E1 -2522.846,E2 -2522.846} C_VEL
LIN {X 0,Y 566.239,Z 377.954,A -85,B 0,C 180,E1 -2525.698,E2 -2525.698} C_VEL
LIN {X 0,Y 566.19,Z 377.95,A -85,B 0,C 180,E1 -2528.566,E2 -2528.566} C_VEL
LIN {X 0,Y 566.198,Z 377.954,A -85,B 0,C 180,E1 -2531.455,E2 -2531.455} C_VEL
LIN {X 0,Y 566.207,Z 377.95,A -85,B 0,C 180,E1 -2534.493,E2 -2534.493} C_VEL
LIN {X 0,Y 566.153,Z 377.956,A -85,B 0,C 180,E1 -2537.333,E2 -2537.333} C_VEL
LIN {X 0,Y 566.154,Z 377.959,A -85,B 0,C 180,E1 -2540.339,E2 -2540.339} C_VEL
LIN {X 0,Y 566.162,Z 377.953,A -85,B 0,C 180,E1 -2542.632,E2 -2542.632} C_VEL
LIN {X 0,Y 566.178,Z 377.962,A -85,B 0,C 180,E1 -2545.751,E2 -2545.751} C_VEL
LIN {X 0,Y 566.14,Z 377.96,A -85,B 0,C 180,E1 -2548.189,E2 -2548.189} C_VEL
LIN {X 0,Y 566.185,Z 377.953,A -85,B 0,C 180,E1 -2551.074,E2 -2551.074} C_VEL
LIN {X 0,Y 566.195,Z 377.958,A -85,B 0,C 180,E1 -2553.957,E2 -2553.957} C_VEL
LIN {X 0,Y 566.142,Z 377.959,A -85,B 0,C 180,E1 -2556.574,E2 -2556.574} C_VEL
LIN {X 0,Y 566.195,Z 377.952,A -85,B 0,C 180,E1 -2559.275,E2 -2559.275} C_VEL
LIN {X 0,Y 566.143,Z 377.961,A -85,B 0,C 180,E1 -2562.094,E2 -2562.094} C_VEL
LIN {X 0,Y 566.161,Z 377.956,A -85,B 0,C 180,E1 -2565.037,E2 -2565.037} C_VEL
LIN {X 0,Y 566.139,Z 377.958,A -85,B 0,C 180,E1 -2568.145,E2 -2568.145} C_VEL
LIN {X 0,Y 566.195,Z 377.951,A -85,B 0,C 180,E1 -2570.724,E2 -2570.724} C_VEL
LIN {X 0,Y 566.132,Z 377.963,A -85,B 0,C 180,E1 -2573.425,E2 -2573.425} C_VEL
LIN {X 0,Y 566.18,Z 377.959,A -85,B 0,C 180,E1 -2576.271,E2 -2576.271} C_VEL
LIN {X 0,Y 566.173,Z 377.957,A -85,B 0,C 180,E1 -2578.927,E2 -2578.927} C_VEL
LIN {X 0,Y 566.137,Z 377.963,A -85,B 0,C 180,E1 -2581.853,E2 -2581.853} C_VEL
LIN {X 0,Y 566.212,Z 378.16,A -85,B 0,C 180,E1 -2582.573,E2 -2582.573} C_VEL
LIN {X 0,Y 567.926,Z 385.981,A -85,B 0,C 180,E1 -2583.545,E2 -2583.545} C_VEL
LIN {X 0,Y 567.717,Z 408.287,A -85,B 0,C 180,E1 -2586.039,E2 -2586.039} C_VEL
LIN {X 0,Y 567.401,Z 431.441,A -85,B 0,C 180,E1 -2588.627,E2 -2588.627} C_VEL
LIN {X 0,Y 566.996,Z 457.816,A -85,B 0,C 180,E1 -2591.574,E2 -2591.574} C_VEL
LIN {X 0,Y 566.68,Z 481.35,A -85,B 0,C 180,E1 -2594.166,E2 -2594.166} C_VEL
LIN {X 0,Y 566.562,Z 497.893,A -85,B 0,C 180,E1 -2595.956,E2 -2595.956} C_VEL
LIN {X 0,Y 567.197,Z 503.704,A -85,B 0,C 180,E1 -2596.063,E2 -2596.063} C_VEL
LIN {X 0,Y 566.949,Z 607.937,A -85,B 0,C 180,E1 -2597.403,E2 -2597.403} C_VEL
LIN {X 0,Y 566.853,Z 621.212,A -85,B 0,C 180,E1 -2597.719,E2 -2597.719} C_VEL
LIN {X 0,Y 566.728,Z 634.148,A -85,B 0,C 180,E1 -2598.179,E2 -2598.179} C_VEL
LIN {X 0,Y 566.613,Z 646.245,A -85,B 0,C 180,E1 -2598.77,E2 -2598.77} C_VEL
LIN {X 0,Y 566.421,Z 658.48,A -85,B 0,C 180,E1 -2599.545,E2 -2599.545} C_VEL
LIN {X 0,Y 566.299,Z 668.645,A -85,B 0,C 180,E1 -2600.355,E2 -2600.355} C_VEL
LIN {X 0,Y 566.166,Z 677.785,A -85,B 0,C 180,E1 -2601.253,E2 -2601.253} C_VEL
LIN {X 0,Y 566.081,Z 686.688,A -85,B 0,C 180,E1 -2602.33,E2 -2602.33} C_VEL
LIN {X 0,Y 565.968,Z 693.955,A -85,B 0,C 180,E1 -2603.422,E2 -2603.422} C_VEL
LIN {X 0,Y 566.004,Z 698.679,A -85,B 0,C 180,E1 -2604.299,E2 -2604.299} C_VEL
LIN {X 0,Y 565.933,Z 703.372,A -85,B 0,C 180,E1 -2605.37,E2 -2605.37} C_VEL
LIN {X 0,Y 565.927,Z 706.957,A -85,B 0,C 180,E1 -2606.44,E2 -2606.44} C_VEL
LIN {X 0,Y 565.878,Z 708.808,A -85,B 0,C 180,E1 -2607.152,E2 -2607.152} C_VEL
LIN {X 0,Y 565.846,Z 711.185,A -85,B 0,C 180,E1 -2608.576,E2 -2608.576} C_VEL
LIN {X 0,Y 565.839,Z 712,A -85,B 0,C 180,E1 -2610,E2 -2610} C_VEL
LIN {X 0,Y 565.846,Z 711.186,A -85,B 0,C 180,E1 -2611.423,E2 -2611.423} C_VEL
LIN {X 0,Y 565.878,Z 708.81,A -85,B 0,C 180,E1 -2612.847,E2 -2612.847} C_VEL
LIN {X 0,Y 565.926,Z 705.896,A -85,B 0,C 180,E1 -2613.916,E2 -2613.916} C_VEL
LIN {X 0,Y 565.878,Z 701.949,A -85,B 0,C 180,E1 -2614.987,E2 -2614.987} C_VEL
LIN {X 0,Y 566.002,Z 696.867,A -85,B 0,C 180,E1 -2616.058,E2 -2616.058} C_VEL
LIN {X 0,Y 566.04,Z 690.469,A -85,B 0,C 180,E1 -2617.132,E2 -2617.132} C_VEL
LIN {X 0,Y 566.134,Z 682.478,A -85,B 0,C 180,E1 -2618.208,E2 -2618.208} C_VEL
LIN {X 0,Y 566.229,Z 674.336,A -85,B 0,C 180,E1 -2619.105,E2 -2619.105} C_VEL
LIN {X 0,Y 566.345,Z 664.401,A -85,B 0,C 180,E1 -2620.005,E2 -2620.005} C_VEL
LIN {X 0,Y 566.544,Z 653.284,A -85,B 0,C 180,E1 -2620.807,E2 -2620.807} C_VEL
LIN {X 0,Y 566.66,Z 642.177,A -85,B 0,C 180,E1 -2621.446,E2 -2621.446} C_VEL
LIN {X 0,Y 566.755,Z 629.984,A -85,B 0,C 180,E1 -2621.988,E2 -2621.988} C_VEL
LIN {X 0,Y 566.896,Z 617.177,A -85,B 0,C 180,E1 -2622.394,E2 -2622.394} C_VEL
LIN {X 0,Y 567.002,Z 603.602,A -85,B 0,C 180,E1 -2622.664,E2 -2622.664} C_VEL
LIN {X 0,Y 567.066,Z 501.929,A -85,B 0,C 180,E1 -2623.963,E2 -2623.963} C_VEL
LIN {X 0,Y 566.561,Z 497.895,A -85,B 0,C 180,E1 -2624.044,E2 -2624.044} C_VEL
LIN {X 0,Y 566.834,Z 471.46,A -85,B 0,C 180,E1 -2626.919,E2 -2626.919} C_VEL
LIN {X 0,Y 567.141,Z 446.22,A -85,B 0,C 180,E1 -2629.717,E2 -2629.717} C_VEL
LIN {X 0,Y 567.566,Z 422.516,A -85,B 0,C 180,E1 -2632.381,E2 -2632.381} C_VEL
LIN {X 0,Y 567.747,Z 398.269,A -85,B 0,C 180,E1 -2635.017,E2 -2635.017} C_VEL
LIN {X 0,Y 567.763,Z 385.004,A -85,B 0,C 180,E1 -2636.463,E2 -2636.463} C_VEL
LIN {X 0,Y 566.179,Z 378.072,A -85,B 0,C 180,E1 -2637.322,E2 -2637.322} C_VEL
LIN {X 0,Y 566.154,Z 377.966,A -85,B 0,C 180,E1 -2639.772,E2 -2639.772} C_VEL
LIN {X 0,Y 566.171,Z 377.959,A -85,B 0,C 180,E1 -2642.424,E2 -2642.424} C_VEL
LIN {X 0,Y 566.157,Z 377.958,A -85,B 0,C 180,E1 -2644.986,E2 -2644.986} C_VEL
LIN {X 0,Y 566.182,Z 377.958,A -85,B 0,C 180,E1 -2647.462,E2 -2647.462} C_VEL
LIN {X 0,Y 566.16,Z 377.961,A -85,B 0,C 180,E1 -2650.203,E2 -2650.203} C_VEL
LIN {X 0,Y 566.147,Z 377.959,A -85,B 0,C 180,E1 -2653.06,E2 -2653.06} C_VEL
LIN {X 0,Y 566.157,Z 377.962,A -85,B 0,C 180,E1 -2656.053,E2 -2656.053} C_VEL
LIN {X 0,Y 566.157,Z 377.957,A -85,B 0,C 180,E1 -2658.859,E2 -2658.859} C_VEL
LIN {X 0,Y 566.203,Z 377.958,A -85,B 0,C 180,E1 -2661.443,E2 -2661.443} C_VEL
LIN {X 0,Y 566.143,Z 377.96,A -85,B 0,C 180,E1 -2664.306,E2 -2664.306} C_VEL
LIN {X 0,Y 566.206,Z 377.952,A -85,B 0,C 180,E1 -2666.897,E2 -2666.897} C_VEL
LIN {X 0,Y 566.18,Z 377.963,A -85,B 0,C 180,E1 -2669.407,E2 -2669.407} C_VEL
LIN {X 0,Y 566.19,Z 377.957,A -85,B 0,C 180,E1 -2671.856,E2 -2671.856} C_VEL
LIN {X 0,Y 566.24,Z 377.95,A -85,B 0,C 180,E1 -2675.039,E2 -2675.039} C_VEL
LIN {X 0,Y 566.195,Z 377.953,A -85,B 0,C 180,E1 -2678.137,E2 -2678.137} C_VEL
LIN {X 0,Y 566.234,Z 377.949,A -85,B 0,C 180,E1 -2680.614,E2 -2680.614} C_VEL
LIN {X 0,Y 566.217,Z 377.959,A -85,B 0,C 180,E1 -2683.412,E2 -2683.412} C_VEL
LIN {X 0,Y 566.277,Z 378.117,A -85,B 0,C 180,E1 -2686.292,E2 -2686.292} C_VEL
LIN {X 0,Y 566.494,Z 379.134,A -85,B 0,C 180,E1 -2686.406,E2 -2686.406} C_VEL
LIN {X 0,Y 567.059,Z 381.003,A -85,B 0,C 180,E1 -2686.454,E2 -2686.454} C_VEL
LIN {X 0,Y 566.993,Z 457.55,A -85,B 0,C 180,E1 -2687.449,E2 -2687.449} C_VEL
LIN {X 0,Y 566.882,Z 467.804,A -85,B 0,C 180,E1 -2687.674,E2 -2687.674} C_VEL
LIN {X 0,Y 566.751,Z 478.576,A -85,B 0,C 180,E1 -2688.012,E2 -2688.012} C_VEL
LIN {X 0,Y 566.68,Z 489.135,A -85,B 0,C 180,E1 -2688.455,E2 -2688.455} C_VEL
LIN {X 0,Y 566.587,Z 499.851,A -85,B 0,C 180,E1 -2689.026,E2 -2689.026} C_VEL
LIN {X 0,Y 566.428,Z 511.518,A -85,B 0,C 180,E1 -2689.816,E2 -2689.816} C_VEL
LIN {X 0,Y 566.306,Z 520.109,A -85,B 0,C 180,E1 -2690.536,E2 -2690.536} C_VEL
LIN {X 0,Y 566.2,Z 528.955,A -85,B 0,C 180,E1 -2691.434,E2 -2691.434} C_VEL
LIN {X 0,Y 566.081,Z 536.289,A -85,B 0,C 180,E1 -2692.33,E2 -2692.33} C_VEL
LIN {X 0,Y 566.018,Z 541.804,A -85,B 0,C 180,E1 -2693.127,E2 -2693.127} C_VEL
LIN {X 0,Y 566.003,Z 546.604,A -85,B 0,C 180,E1 -2693.942,E2 -2693.942} C_VEL
LIN {X 0,Y 565.877,Z 551.716,A -85,B 0,C 180,E1 -2695.013,E2 -2695.013} C_VEL
LIN {X 0,Y 565.926,Z 555.698,A -85,B 0,C 180,E1 -2696.084,E2 -2696.084} C_VEL
LIN {X 0,Y 565.877,Z 558.65,A -85,B 0,C 180,E1 -2697.152,E2 -2697.152} C_VEL
LIN {X 0,Y 565.84,Z 560.135,A -85,B 0,C 180,E1 -2697.865,E2 -2697.865} C_VEL
LIN {X 0,Y 565.841,Z 561.724,A -85,B 0,C 180,E1 -2699.288,E2 -2699.288} C_VEL
LIN {X 0,Y 565.839,Z 561.996,A -85,B 0,C 180,E1 -2700,E2 -2700} C_VEL
LIN {X 0,Y 565.846,Z 561.213,A -85,B 0,C 180,E1 -2701.423,E2 -2701.423} C_VEL
LIN {X 0,Y 565.84,Z 560.281,A -85,B 0,C 180,E1 -2702.135,E2 -2702.135} C_VEL
LIN {X 0,Y 565.927,Z 557.057,A -85,B 0,C 180,E1 -2703.56,E2 -2703.56} C_VEL
LIN {X 0,Y 565.933,Z 553.499,A -85,B 0,C 180,E1 -2704.63,E2 -2704.63} C_VEL
LIN {X 0,Y 565.998,Z 548.844,A -85,B 0,C 180,E1 -2705.701,E2 -2705.701} C_VEL
LIN {X 0,Y 565.996,Z 543.172,A -85,B 0,C 180,E1 -2706.739,E2 -2706.739} C_VEL
LIN {X 0,Y 566.081,Z 536.947,A -85,B 0,C 180,E1 -2707.67,E2 -2707.67} C_VEL
LIN {X 0,Y 566.17,Z 529.735,A -85,B 0,C 180,E1 -2708.567,E2 -2708.567} C_VEL
LIN {X 0,Y 566.249,Z 522.892,A -85,B 0,C 180,E1 -2709.285,E2 -2709.285} C_VEL
LIN {X 0,Y 566.344,Z 514.829,A -85,B 0,C 180,E1 -2710.005,E2 -2710.005} C_VEL
LIN {X 0,Y 566.459,Z 506.448,A -85,B 0,C 180,E1 -2710.635,E2 -2710.635} C_VEL
LIN {X 0,Y 566.569,Z 498.355,A -85,B 0,C 180,E1 -2711.149,E2 -2711.149} C_VEL
LIN {X 0,Y 566.686,Z 488.641,A -85,B 0,C 180,E1 -2711.658,E2 -2711.658} C_VEL
LIN {X 0,Y 566.768,Z 478.554,A -85,B 0,C 180,E1 -2712.079,E2 -2712.079} C_VEL
LIN {X 0,Y 566.877,Z 467.768,A -85,B 0,C 180,E1 -2712.417,E2 -2712.417} C_VEL
LIN {X 0,Y 566.977,Z 457.535,A -85,B 0,C 180,E1 -2712.642,E2 -2712.642} C_VEL
LIN {X 0,Y 566.992,Z 380.804,A -85,B 0,C 180,E1 -2713.641,E2 -2713.641} C_VEL
LIN {X 0,Y 566.412,Z 378.807,A -85,B 0,C 180,E1 -2713.705,E2 -2713.705} C_VEL
LIN {X 0,Y 566.254,Z 377.999,A -85,B 0,C 180,E1 -2713.846,E2 -2713.846} C_VEL
LIN {X 0,Y 566.216,Z 377.957,A -85,B 0,C 180,E1 -2716.616,E2 -2716.616} C_VEL
LIN {X 0,Y 565.555,Z 378.038,A -85,B 0,C 180,E1 -2717.209,E2 -2717.209} C_VEL
LIN {X 0,Y 562.721,Z 378.388,A -85,B 0,C 180,E1 -2718.172,E2 -2718.172} C_VEL
LIN {X 0,Y 560.316,Z 378.693,A -85,B 0,C 180,E1 -2718.947,E2 -2718.947} C_VEL
LIN {X 0,Y 559.268,Z 378.817,A -85,B 0,C 180,E1 -2719.545,E2 -2719.545} C_VEL
LIN {X 0,Y 559.175,Z 378.827,A -85,B 0,C 180,E1 -2719.748,E2 -2719.748} C_VEL
LIN {X 0,Y 559.144,Z 378.832,A -85,B 0,C 180,E1 -2722.153,E2 -2722.153} C_VEL
LIN {X 0,Y 559.178,Z 378.828,A -85,B 0,C 180,E1 -2725.298,E2 -2725.298} C_VEL
LIN {X 0,Y 559.132,Z 378.83,A -85,B 0,C 180,E1 -2727.715,E2 -2727.715} C_VEL
LIN {X 0,Y 559.156,Z 378.829,A -85,B 0,C 180,E1 -2730.183,E2 -2730.183} C_VEL
LIN {X 0,Y 559.155,Z 378.837,A -85,B 0,C 180,E1 -2732.715,E2 -2732.715} C_VEL
LIN {X 0,Y 559.127,Z 378.834,A -85,B 0,C 180,E1 -2735.324,E2 -2735.324} C_VEL
LIN {X 0,Y 559.134,Z 378.831,A -85,B 0,C 180,E1 -2738.018,E2 -2738.018} C_VEL
LIN {X 0,Y 559.158,Z 378.835,A -85,B 0,C 180,E1 -2740.813,E2 -2740.813} C_VEL
LIN {X 0,Y 559.113,Z 378.835,A -85,B 0,C 180,E1 -2743.737,E2 -2743.737} C_VEL
LIN {X 0,Y 559.139,Z 378.835,A -85,B 0,C 180,E1 -2746.266,E2 -2746.266} C_VEL
LIN {X 0,Y 559.158,Z 378.831,A -85,B 0,C 180,E1 -2749.188,E2 -2749.188} C_VEL
LIN {X 0,Y 559.131,Z 378.83,A -85,B 0,C 180,E1 -2751.982,E2 -2751.982} C_VEL
LIN {X 0,Y 559.13,Z 378.837,A -85,B 0,C 180,E1 -2754.788,E2 -2754.788} C_VEL
LIN {X 0,Y 559.158,Z 378.828,A -85,B 0,C 180,E1 -2757.365,E2 -2757.365} C_VEL
LIN {X 0,Y 559.145,Z 378.835,A -85,B 0,C 180,E1 -2760.144,E2 -2760.144} C_VEL
LIN {X 0,Y 559.163,Z 378.979,A -85,B 0,C 180,E1 -2763.022,E2 -2763.022} C_VEL
LIN {X 0,Y 560.869,Z 387.666,A -85,B 0,C 180,E1 -2764.132,E2 -2764.132} C_VEL
LIN {X 0,Y 560.609,Z 413.369,A -85,B 0,C 180,E1 -2767.131,E2 -2767.131} C_VEL
LIN {X 0,Y 560.289,Z 436.494,A -85,B 0,C 180,E1 -2769.821,E2 -2769.821} C_VEL
LIN {X 0,Y 559.829,Z 461.083,A -85,B 0,C 180,E1 -2772.704,E2 -2772.704} C_VEL
LIN {X 0,Y 559.579,Z 486.416,A -85,B 0,C 180,E1 -2775.638,E2 -2775.638} C_VEL
LIN {X 0,Y 559.576,Z 488.235,A -85,B 0,C 180,E1 -2775.823,E2 -2775.823} C_VEL
LIN {X 0,Y 560.297,Z 495.609,A -85,B 0,C 180,E1 -2775.958,E2 -2775.958} C_VEL
LIN {X 0,Y 560.044,Z 597.966,A -85,B 0,C 180,E1 -2777.291,E2 -2777.291} C_VEL
LIN {X 0,Y 559.964,Z 609.557,A -85,B 0,C 180,E1 -2777.565,E2 -2777.565} C_VEL
LIN {X 0,Y 559.801,Z 619.857,A -85,B 0,C 180,E1 -2777.907,E2 -2777.907} C_VEL
LIN {X 0,Y 559.724,Z 629.931,A -85,B 0,C 180,E1 -2778.347,E2 -2778.347} C_VEL
LIN {X 0,Y 559.602,Z 640.07,A -85,B 0,C 180,E1 -2778.903,E2 -2778.903} C_VEL
LIN {X 0,Y 559.437,Z 650.295,A -85,B 0,C 180,E1 -2779.596,E2 -2779.596} C_VEL
LIN {X 0,Y 559.278,Z 660.145,A -85,B 0,C 180,E1 -2780.416,E2 -2780.416} C_VEL
LIN {X 0,Y 559.14,Z 669.032,A -85,B 0,C 180,E1 -2781.325,E2 -2781.325} C_VEL
LIN {X 0,Y 558.997,Z 677.625,A -85,B 0,C 180,E1 -2782.414,E2 -2782.414} C_VEL
LIN {X 0,Y 558.946,Z 683.844,A -85,B 0,C 180,E1 -2783.376,E2 -2783.376} C_VEL
LIN {X 0,Y 558.936,Z 688.424,A -85,B 0,C 180,E1 -2784.227,E2 -2784.227} C_VEL
LIN {X 0,Y 558.826,Z 693.156,A -85,B 0,C 180,E1 -2785.311,E2 -2785.311} C_VEL
LIN {X 0,Y 558.836,Z 696.786,A -85,B 0,C 180,E1 -2786.395,E2 -2786.395} C_VEL
LIN {X 0,Y 558.799,Z 698.678,A -85,B 0,C 180,E1 -2787.116,E2 -2787.116} C_VEL
LIN {X 0,Y 558.746,Z 700.139,A -85,B 0,C 180,E1 -2787.838,E2 -2787.838} C_VEL
LIN {X 0,Y 558.741,Z 701.744,A -85,B 0,C 180,E1 -2789.279,E2 -2789.279} C_VEL
LIN {X 0,Y 558.74,Z 701.996,A -85,B 0,C 180,E1 -2790,E2 -2790} C_VEL
LIN {X 0,Y 558.746,Z 701.221,A -85,B 0,C 180,E1 -2791.442,E2 -2791.442} C_VEL
LIN {X 0,Y 558.746,Z 700.282,A -85,B 0,C 180,E1 -2792.163,E2 -2792.163} C_VEL
LIN {X 0,Y 558.836,Z 697.049,A -85,B 0,C 180,E1 -2793.605,E2 -2793.605} C_VEL
LIN {X 0,Y 558.827,Z 693.5,A -85,B 0,C 180,E1 -2794.689,E2 -2794.689} C_VEL
LIN {X 0,Y 558.928,Z 688.856,A -85,B 0,C 180,E1 -2795.773,E2 -2795.773} C_VEL
LIN {X 0,Y 558.929,Z 682.016,A -85,B 0,C 180,E1 -2797.024,E2 -2797.024} C_VEL
LIN {X 0,Y 559.04,Z 674.303,A -85,B 0,C 180,E1 -2798.131,E2 -2798.131} C_VEL
LIN {X 0,Y 559.172,Z 666.499,A -85,B 0,C 180,E1 -2799.039,E2 -2799.039} C_VEL
LIN {X 0,Y 559.294,Z 658.045,A -85,B 0,C 180,E1 -2799.858,E2 -2799.858} C_VEL
LIN {X 0,Y 559.431,Z 649.015,A -85,B 0,C 180,E1 -2800.587,E2 -2800.587} C_VEL
LIN {X 0,Y 559.62,Z 639.172,A -85,B 0,C 180,E1 -2801.241,E2 -2801.241} C_VEL
LIN {X 0,Y 559.694,Z 630.031,A -85,B 0,C 180,E1 -2801.739,E2 -2801.739} C_VEL
LIN {X 0,Y 559.811,Z 620.147,A -85,B 0,C 180,E1 -2802.171,E2 -2802.171} C_VEL
LIN {X 0,Y 559.929,Z 608.705,A -85,B 0,C 180,E1 -2802.551,E2 -2802.551} C_VEL
LIN {X 0,Y 560.093,Z 596.592,A -85,B 0,C 180,E1 -2802.823,E2 -2802.823} C_VEL
LIN {X 0,Y 560.193,Z 492.71,A -85,B 0,C 180,E1 -2804.172,E2 -2804.172} C_VEL
LIN {X 0,Y 559.597,Z 488.133,A -85,B 0,C 180,E1 -2804.269,E2 -2804.269} C_VEL
LIN {X 0,Y 559.873,Z 460.593,A -85,B 0,C 180,E1 -2807.442,E2 -2807.442} C_VEL
LIN {X 0,Y 560.295,Z 435.639,A -85,B 0,C 180,E1 -2810.37,E2 -2810.37} C_VEL
LIN {X 0,Y 560.632,Z 412.507,A -85,B 0,C 180,E1 -2813.063,E2 -2813.063} C_VEL
LIN {X 0,Y 560.874,Z 387.213,A -85,B 0,C 180,E1 -2816.013,E2 -2816.013} C_VEL
LIN {X 0,Y 559.158,Z 378.946,A -85,B 0,C 180,E1 -2817.08,E2 -2817.08} C_VEL
LIN {X 0,Y 559.14,Z 378.835,A -85,B 0,C 180,E1 -2820.184,E2 -2820.184} C_VEL
LIN {X 0,Y 559.154,Z 378.83,A -85,B 0,C 180,E1 -2822.716,E2 -2822.716} C_VEL
LIN {X 0,Y 559.12,Z 378.839,A -85,B 0,C 180,E1 -2825.325,E2 -2825.325} C_VEL
LIN {X 0,Y 559.127,Z 378.837,A -85,B 0,C 180,E1 -2828.018,E2 -2828.018} C_VEL
LIN {X 0,Y 559.161,Z 378.831,A -85,B 0,C 180,E1 -2829.941,E2 -2829.941} C_VEL
LIN {X 0,Y 559.117,Z 378.834,A -85,B 0,C 180,E1 -2832.748,E2 -2832.748} C_VEL
LIN {X 0,Y 559.127,Z 378.839,A -85,B 0,C 180,E1 -2835.764,E2 -2835.764} C_VEL
LIN {X 0,Y 559.127,Z 378.834,A -85,B 0,C 180,E1 -2838.226,E2 -2838.226} C_VEL
LIN {X 0,Y 559.172,Z 378.83,A -85,B 0,C 180,E1 -2841.193,E2 -2841.193} C_VEL
LIN {X 0,Y 559.118,Z 378.842,A -85,B 0,C 180,E1 -2843.787,E2 -2843.787} C_VEL
LIN {X 0,Y 559.149,Z 378.828,A -85,B 0,C 180,E1 -2846.424,E2 -2846.424} C_VEL
LIN {X 0,Y 559.153,Z 378.83,A -85,B 0,C 180,E1 -2848.98,E2 -2848.98} C_VEL
LIN {X 0,Y 559.112,Z 378.841,A -85,B 0,C 180,E1 -2851.631,E2 -2851.631} C_VEL
LIN {X 0,Y 559.129,Z 378.832,A -85,B 0,C 180,E1 -2854.699,E2 -2854.699} C_VEL
LIN {X 0,Y 559.12,Z 378.832,A -85,B 0,C 180,E1 -2857.066,E2 -2857.066} C_VEL
LIN {X 0,Y 559.167,Z 378.832,A -85,B 0,C 180,E1 -2859.395,E2 -2859.395} C_VEL
LIN {X 0,Y 559.122,Z 378.839,A -85,B 0,C 180,E1 -2861.685,E2 -2861.685} C_VEL
LIN {X 0,Y 559.136,Z 378.831,A -85,B 0,C 180,E1 -2864.695,E2 -2864.695} C_VEL
LIN {X 0,Y 559.174,Z 378.834,A -85,B 0,C 180,E1 -2867.663,E2 -2867.663} C_VEL
LIN {X 0,Y 559.137,Z 378.83,A -85,B 0,C 180,E1 -2870.596,E2 -2870.596} C_VEL
LIN {X 0,Y 559.148,Z 378.835,A -85,B 0,C 180,E1 -2873.505,E2 -2873.505} C_VEL
LIN {X 0,Y 559.131,Z 378.836,A -85,B 0,C 180,E1 -2875.675,E2 -2875.675} C_VEL
LIN {X 0,Y 559.25,Z 378.826,A -85,B 0,C 180,E1 -2877.839,E2 -2877.839} C_VEL
LIN {X 0,Y 559.257,Z 378.821,A -85,B 0,C 180,E1 -2880,E2 -2880} C_VEL
LIN {X 0,Y 559.21,Z 378.817,A -85,B 0,C 180,E1 -2882.882,E2 -2882.882} C_VEL
LIN {X 0,Y 559.208,Z 378.832,A -85,B 0,C 180,E1 -2885.77,E2 -2885.77} C_VEL
LIN {X 0,Y 559.155,Z 378.826,A -85,B 0,C 180,E1 -2888.675,E2 -2888.675} C_VEL
LIN {X 0,Y 559.16,Z 378.832,A -85,B 0,C 180,E1 -2891.601,E2 -2891.601} C_VEL
LIN {X 0,Y 559.157,Z 378.828,A -85,B 0,C 180,E1 -2894.576,E2 -2894.576} C_VEL
LIN {X 0,Y 559.11,Z 378.836,A -85,B 0,C 180,E1 -2897.559,E2 -2897.559} C_VEL
LIN {X 0,Y 559.114,Z 378.834,A -85,B 0,C 180,E1 -2900.607,E2 -2900.607} C_VEL
LIN {X 0,Y 559.135,Z 378.831,A -85,B 0,C 180,E1 -2903.426,E2 -2903.426} C_VEL
LIN {X 0,Y 559.146,Z 378.835,A -85,B 0,C 180,E1 -2906.099,E2 -2906.099} C_VEL
LIN {X 0,Y 559.101,Z 378.833,A -85,B 0,C 180,E1 -2908.533,E2 -2908.533} C_VEL
LIN {X 0,Y 559.14,Z 378.832,A -85,B 0,C 180,E1 -2911.271,E2 -2911.271} C_VEL
LIN {X 0,Y 559.153,Z 378.835,A -85,B 0,C 180,E1 -2913.946,E2 -2913.946} C_VEL
LIN {X 0,Y 559.112,Z 378.835,A -85,B 0,C 180,E1 -2917.111,E2 -2917.111} C_VEL
LIN {X 0,Y 559.12,Z 378.834,A -85,B 0,C 180,E1 -2919.936,E2 -2919.936} C_VEL
LIN {X 0,Y 559.11,Z 378.83,A -85,B 0,C 180,E1 -2922.748,E2 -2922.748} C_VEL
LIN {X 0,Y 559.123,Z 378.841,A -85,B 0,C 180,E1 -2925.764,E2 -2925.764} C_VEL
LIN {X 0,Y 559.096,Z 378.833,A -85,B 0,C 180,E1 -2928.223,E2 -2928.223} C_VEL
LIN {X 0,Y 559.138,Z 378.831,A -85,B 0,C 180,E1 -2931.197,E2 -2931.197} C_VEL
LIN {X 0,Y 559.108,Z 378.843,A -85,B 0,C 180,E1 -2933.786,E2 -2933.786} C_VEL
LIN {X 0,Y 559.125,Z 378.836,A -85,B 0,C 180,E1 -2936.422,E2 -2936.422} C_VEL
LIN {X 0,Y 559.139,Z 378.833,A -85,B 0,C 180,E1 -2938.979,E2 -2938.979} C_VEL
LIN {X 0,Y 559.146,Z 378.96,A -85,B 0,C 180,E1 -2942.352,E2 -2942.352} C_VEL
LIN {X 0,Y 561.029,Z 387.115,A -85,B 0,C 180,E1 -2943.395,E2 -2943.395} C_VEL
LIN {X 0,Y 560.866,Z 408.113,A -85,B 0,C 180,E1 -2945.775,E2 -2945.775} C_VEL
LIN {X 0,Y 560.481,Z 434.142,A -85,B 0,C 180,E1 -2948.676,E2 -2948.676} C_VEL
LIN {X 0,Y 560.072,Z 459.497,A -85,B 0,C 180,E1 -2951.527,E2 -2951.527} C_VEL
LIN {X 0,Y 559.727,Z 483.031,A -85,B 0,C 180,E1 -2954.151,E2 -2954.151} C_VEL
LIN {X 0,Y 559.604,Z 497.897,A -85,B 0,C 180,E1 -2955.778,E2 -2955.778} C_VEL
LIN {X 0,Y 560.328,Z 505.493,A -85,B 0,C 180,E1 -2955.912,E2 -2955.912} C_VEL
LIN {X 0,Y 560.028,Z 607.937,A -85,B 0,C 180,E1 -2957.244,E2 -2957.244} C_VEL
LIN {X 0,Y 559.919,Z 621.212,A -85,B 0,C 180,E1 -2957.564,E2 -2957.564} C_VEL
LIN {X 0,Y 559.792,Z 634.15,A -85,B 0,C 180,E1 -2958.031,E2 -2958.031} C_VEL
LIN {X 0,Y 559.634,Z 646.845,A -85,B 0,C 180,E1 -2958.663,E2 -2958.663} C_VEL
LIN {X 0,Y 559.437,Z 658.481,A -85,B 0,C 180,E1 -2959.413,E2 -2959.413} C_VEL
LIN {X 0,Y 559.296,Z 668.645,A -85,B 0,C 180,E1 -2960.233,E2 -2960.233} C_VEL
LIN {X 0,Y 559.134,Z 677.785,A -85,B 0,C 180,E1 -2961.142,E2 -2961.142} C_VEL
LIN {X 0,Y 559.01,Z 686.688,A -85,B 0,C 180,E1 -2962.232,E2 -2962.232} C_VEL
LIN {X 0,Y 558.925,Z 692.74,A -85,B 0,C 180,E1 -2963.14,E2 -2963.14} C_VEL
LIN {X 0,Y 558.935,Z 698.679,A -85,B 0,C 180,E1 -2964.227,E2 -2964.227} C_VEL
LIN {X 0,Y 558.826,Z 703.372,A -85,B 0,C 180,E1 -2965.311,E2 -2965.311} C_VEL
LIN {X 0,Y 558.836,Z 706.957,A -85,B 0,C 180,E1 -2966.395,E2 -2966.395} C_VEL
LIN {X 0,Y 558.799,Z 708.807,A -85,B 0,C 180,E1 -2967.116,E2 -2967.116} C_VEL
LIN {X 0,Y 558.745,Z 711.185,A -85,B 0,C 180,E1 -2968.558,E2 -2968.558} C_VEL
LIN {X 0,Y 558.74,Z 712,A -85,B 0,C 180,E1 -2970,E2 -2970} C_VEL
LIN {X 0,Y 558.745,Z 711.186,A -85,B 0,C 180,E1 -2971.441,E2 -2971.441} C_VEL
LIN {X 0,Y 558.799,Z 708.81,A -85,B 0,C 180,E1 -2972.884,E2 -2972.884} C_VEL
LIN {X 0,Y 558.844,Z 705.896,A -85,B 0,C 180,E1 -2973.966,E2 -2973.966} C_VEL
LIN {X 0,Y 558.798,Z 701.949,A -85,B 0,C 180,E1 -2975.051,E2 -2975.051} C_VEL
LIN {X 0,Y 558.921,Z 696.867,A -85,B 0,C 180,E1 -2976.135,E2 -2976.135} C_VEL
LIN {X 0,Y 558.977,Z 690.468,A -85,B 0,C 180,E1 -2977.223,E2 -2977.223} C_VEL
LIN {X 0,Y 559.099,Z 682.478,A -85,B 0,C 180,E1 -2978.312,E2 -2978.312} C_VEL
LIN {X 0,Y 559.185,Z 674.335,A -85,B 0,C 180,E1 -2979.221,E2 -2979.221} C_VEL
LIN {X 0,Y 559.356,Z 664.4,A -85,B 0,C 180,E1 -2980.131,E2 -2980.131} C_VEL
LIN {X 0,Y 559.558,Z 653.365,A -85,B 0,C 180,E1 -2980.939,E2 -2980.939} C_VEL
LIN {X 0,Y 559.703,Z 641.142,A -85,B 0,C 180,E1 -2981.644,E2 -2981.644} C_VEL
LIN {X 0,Y 559.842,Z 628.768,A -85,B 0,C 180,E1 -2982.184,E2 -2982.184} C_VEL
LIN {X 0,Y 559.965,Z 615.347,A -85,B 0,C 180,E1 -2982.596,E2 -2982.596} C_VEL
LIN {X 0,Y 560.134,Z 602.085,A -85,B 0,C 180,E1 -2982.845,E2 -2982.845} C_VEL
LIN {X 0,Y 560.194,Z 502.603,A -85,B 0,C 180,E1 -2984.129,E2 -2984.129} C_VEL
LIN {X 0,Y 559.601,Z 497.901,A -85,B 0,C 180,E1 -2984.222,E2 -2984.222} C_VEL
LIN {X 0,Y 559.919,Z 469.745,A -85,B 0,C 180,E1 -2987.326,E2 -2987.326} C_VEL
LIN {X 0,Y 560.362,Z 442.69,A -85,B 0,C 180,E1 -2990.367,E2 -2990.367} C_VEL
LIN {X 0,Y 560.601,Z 419.838,A -85,B 0,C 180,E1 -2992.869,E2 -2992.869} C_VEL
LIN {X 0,Y 560.834,Z 395.352,A -85,B 0,C 180,E1 -2995.543,E2 -2995.543} C_VEL
LIN {X 0,Y 560.866,Z 387.502,A -85,B 0,C 180,E1 -2996.413,E2 -2996.413} C_VEL
LIN {X 0,Y 559.139,Z 378.949,A -85,B 0,C 180,E1 -2997.473,E2 -2997.473} C_VEL
LIN {X 0,Y 559.099,Z 378.845,A -85,B 0,C 180,E1 -3000.186,E2 -3000.186} C_VEL
LIN {X 0,Y 559.133,Z 378.834,A -85,B 0,C 180,E1 -3002.717,E2 -3002.717} C_VEL
LIN {X 0,Y 559.112,Z 378.838,A -85,B 0,C 180,E1 -3005.325,E2 -3005.325} C_VEL
LIN {X 0,Y 559.116,Z 378.842,A -85,B 0,C 180,E1 -3008.019,E2 -3008.019} C_VEL
LIN {X 0,Y 559.093,Z 378.837,A -85,B 0,C 180,E1 -3010.818,E2 -3010.818} C_VEL
LIN {X 0,Y 559.101,Z 378.845,A -85,B 0,C 180,E1 -3013.738,E2 -3013.738} C_VEL
LIN {X 0,Y 559.108,Z 378.837,A -85,B 0,C 180,E1 -3016.263,E2 -3016.263} C_VEL
LIN {X 0,Y 559.119,Z 378.834,A -85,B 0,C 180,E1 -3018.955,E2 -3018.955} C_VEL
LIN {X 0,Y 559.17,Z 378.83,A -85,B 0,C 180,E1 -3021.193,E2 -3021.193} C_VEL
LIN {X 0,Y 559.118,Z 378.841,A -85,B 0,C 180,E1 -3023.787,E2 -3023.787} C_VEL
LIN {X 0,Y 559.15,Z 378.831,A -85,B 0,C 180,E1 -3026.424,E2 -3026.424} C_VEL
LIN {X 0,Y 559.155,Z 378.832,A -85,B 0,C 180,E1 -3028.981,E2 -3028.981} C_VEL
LIN {X 0,Y 559.137,Z 378.839,A -85,B 0,C 180,E1 -3031.625,E2 -3031.625} C_VEL
LIN {X 0,Y 559.164,Z 378.83,A -85,B 0,C 180,E1 -3034.817,E2 -3034.817} C_VEL
LIN {X 0,Y 559.143,Z 378.834,A -85,B 0,C 180,E1 -3037.847,E2 -3037.847} C_VEL
LIN {X 0,Y 559.196,Z 378.826,A -85,B 0,C 180,E1 -3040.494,E2 -3040.494} C_VEL
LIN {X 0,Y 559.184,Z 378.835,A -85,B 0,C 180,E1 -3043.198,E2 -3043.198} C_VEL
LIN {X 0,Y 559.239,Z 378.954,A -85,B 0,C 180,E1 -3046.116,E2 -3046.116} C_VEL
LIN {X 0,Y 559.459,Z 380.045,A -85,B 0,C 180,E1 -3046.244,E2 -3046.244} C_VEL
LIN {X 0,Y 560.248,Z 383.15,A -85,B 0,C 180,E1 -3046.315,E2 -3046.315} C_VEL
LIN {X 0,Y 560.081,Z 457.468,A -85,B 0,C 180,E1 -3047.292,E2 -3047.292} C_VEL
LIN {X 0,Y 559.947,Z 467.88,A -85,B 0,C 180,E1 -3047.519,E2 -3047.519} C_VEL
LIN {X 0,Y 559.845,Z 477.432,A -85,B 0,C 180,E1 -3047.816,E2 -3047.816} C_VEL
LIN {X 0,Y 559.776,Z 486.79,A -85,B 0,C 180,E1 -3048.196,E2 -3048.196} C_VEL
LIN {X 0,Y 559.616,Z 497.507,A -85,B 0,C 180,E1 -3048.744,E2 -3048.744} C_VEL
LIN {X 0,Y 559.445,Z 507.829,A -85,B 0,C 180,E1 -3049.413,E2 -3049.413} C_VEL
LIN {X 0,Y 559.293,Z 518.118,A -85,B 0,C 180,E1 -3050.233,E2 -3050.233} C_VEL
LIN {X 0,Y 559.141,Z 527.382,A -85,B 0,C 180,E1 -3051.143,E2 -3051.143} C_VEL
LIN {X 0,Y 559.053,Z 534.967,A -85,B 0,C 180,E1 -3052.051,E2 -3052.051} C_VEL
LIN {X 0,Y 558.967,Z 541.415,A -85,B 0,C 180,E1 -3052.977,E2 -3052.977} C_VEL
LIN {X 0,Y 558.922,Z 546.601,A -85,B 0,C 180,E1 -3053.864,E2 -3053.864} C_VEL
LIN {X 0,Y 558.798,Z 551.71,A -85,B 0,C 180,E1 -3054.949,E2 -3054.949} C_VEL
LIN {X 0,Y 558.844,Z 555.689,A -85,B 0,C 180,E1 -3056.034,E2 -3056.034} C_VEL
LIN {X 0,Y 558.799,Z 558.64,A -85,B 0,C 180,E1 -3057.116,E2 -3057.116} C_VEL
LIN {X 0,Y 558.746,Z 560.135,A -85,B 0,C 180,E1 -3057.837,E2 -3057.837} C_VEL
LIN {X 0,Y 558.741,Z 561.714,A -85,B 0,C 180,E1 -3059.279,E2 -3059.279} C_VEL
LIN {X 0,Y 558.74,Z 561.996,A -85,B 0,C 180,E1 -3060,E2 -3060} C_VEL
LIN {X 0,Y 558.746,Z 561.201,A -85,B 0,C 180,E1 -3061.442,E2 -3061.442} C_VEL
LIN {X 0,Y 558.746,Z 560.281,A -85,B 0,C 180,E1 -3062.163,E2 -3062.163} C_VEL
LIN {X 0,Y 558.836,Z 557.046,A -85,B 0,C 180,E1 -3063.605,E2 -3063.605} C_VEL
LIN {X 0,Y 558.826,Z 553.488,A -85,B 0,C 180,E1 -3064.689,E2 -3064.689} C_VEL
LIN {X 0,Y 558.928,Z 548.831,A -85,B 0,C 180,E1 -3065.773,E2 -3065.773} C_VEL
LIN {X 0,Y 558.926,Z 542.94,A -85,B 0,C 180,E1 -3066.86,E2 -3066.86} C_VEL
LIN {X 0,Y 559.008,Z 536.929,A -85,B 0,C 180,E1 -3067.767,E2 -3067.767} C_VEL
LIN {X 0,Y 559.101,Z 529.715,A -85,B 0,C 180,E1 -3068.676,E2 -3068.676} C_VEL
LIN {X 0,Y 559.223,Z 522.869,A -85,B 0,C 180,E1 -3069.403,E2 -3069.403} C_VEL
LIN {X 0,Y 559.342,Z 514.869,A -85,B 0,C 180,E1 -3070.131,E2 -3070.131} C_VEL
LIN {X 0,Y 559.514,Z 505.176,A -85,B 0,C 180,E1 -3070.86,E2 -3070.86} C_VEL
LIN {X 0,Y 559.688,Z 493.117,A -85,B 0,C 180,E1 -3071.59,E2 -3071.59} C_VEL
LIN {X 0,Y 559.835,Z 480.274,A -85,B 0,C 180,E1 -3072.171,E2 -3072.171} C_VEL
LIN {X 0,Y 559.96,Z 468.659,A -85,B 0,C 180,E1 -3072.55,E2 -3072.55} C_VEL
LIN {X 0,Y 560.058,Z 458.752,A -85,B 0,C 180,E1 -3072.778,E2 -3072.778} C_VEL
LIN {X 0,Y 560.183,Z 421.383,A -85,B 0,C 180,E1 -3073.282,E2 -3073.282} C_VEL
LIN {X 0,Y 560.102,Z 382.139,A -85,B 0,C 180,E1 -3073.793,E2 -3073.793} C_VEL
LIN {X 0,Y 559.341,Z 379.519,A -85,B 0,C 180,E1 -3073.881,E2 -3073.881} C_VEL
LIN {X 0,Y 559.214,Z 378.85,A -85,B 0,C 180,E1 -3074.047,E2 -3074.047} C_VEL
LIN {X 0,Y 559.175,Z 378.832,A -85,B 0,C 180,E1 -3077.213,E2 -3077.213} C_VEL
LIN {X 0,Y 559.175,Z 378.827,A -85,B 0,C 180,E1 -3079.748,E2 -3079.748} C_VEL
LIN {X 0,Y 558.481,Z 378.918,A -85,B 0,C 180,E1 -3080.349,E2 -3080.349} C_VEL
LIN {X 0,Y 555.601,Z 379.275,A -85,B 0,C 180,E1 -3081.324,E2 -3081.324} C_VEL
LIN {X 0,Y 553.187,Z 379.575,A -85,B 0,C 180,E1 -3082.11,E2 -3082.11} C_VEL
LIN {X 0,Y 552.163,Z 379.709,A -85,B 0,C 180,E1 -3082.716,E2 -3082.716} C_VEL
LIN {X 0,Y 552.085,Z 379.712,A -85,B 0,C 180,E1 -3082.921,E2 -3082.921} C_VEL
LIN {X 0,Y 552.13,Z 379.704,A -85,B 0,C 180,E1 -3085.644,E2 -3085.644} C_VEL
LIN {X 0,Y 552.101,Z 379.713,A -85,B 0,C 180,E1 -3088.557,E2 -3088.557} C_VEL
LIN {X 0,Y 552.114,Z 379.707,A -85,B 0,C 180,E1 -3091.476,E2 -3091.476} C_VEL
LIN {X 0,Y 552.129,Z 379.703,A -85,B 0,C 180,E1 -3094.169,E2 -3094.169} C_VEL
LIN {X 0,Y 552.101,Z 379.715,A -85,B 0,C 180,E1 -3096.748,E2 -3096.748} C_VEL
LIN {X 0,Y 552.131,Z 379.704,A -85,B 0,C 180,E1 -3099.527,E2 -3099.527} C_VEL
LIN {X 0,Y 552.112,Z 379.712,A -85,B 0,C 180,E1 -3102.427,E2 -3102.427} C_VEL
LIN {X 0,Y 552.094,Z 379.708,A -85,B 0,C 180,E1 -3105.562,E2 -3105.562} C_VEL
LIN {X 0,Y 552.123,Z 379.714,A -85,B 0,C 180,E1 -3108.679,E2 -3108.679} C_VEL
LIN {X 0,Y 552.117,Z 379.702,A -85,B 0,C 180,E1 -3111.411,E2 -3111.411} C_VEL
LIN {X 0,Y 552.077,Z 379.715,A -85,B 0,C 180,E1 -3114.156,E2 -3114.156} C_VEL
LIN {X 0,Y 552.118,Z 379.71,A -85,B 0,C 180,E1 -3116.814,E2 -3116.814} C_VEL
LIN {X 0,Y 552.1,Z 379.709,A -85,B 0,C 180,E1 -3119.39,E2 -3119.39} C_VEL
LIN {X 0,Y 552.081,Z 379.714,A -85,B 0,C 180,E1 -3121.9,E2 -3121.9} C_VEL
LIN {X 0,Y 552.155,Z 379.888,A -85,B 0,C 180,E1 -3122.837,E2 -3122.837} C_VEL
LIN {X 0,Y 553.99,Z 388.878,A -85,B 0,C 180,E1 -3124.002,E2 -3124.002} C_VEL
LIN {X 0,Y 553.712,Z 414.582,A -85,B 0,C 180,E1 -3127.027,E2 -3127.027} C_VEL
LIN {X 0,Y 553.308,Z 439.513,A -85,B 0,C 180,E1 -3129.943,E2 -3129.943} C_VEL
LIN {X 0,Y 552.871,Z 464.386,A -85,B 0,C 180,E1 -3132.87,E2 -3132.87} C_VEL
LIN {X 0,Y 552.608,Z 488.26,A -85,B 0,C 180,E1 -3135.641,E2 -3135.641} C_VEL
LIN {X 0,Y 553.435,Z 495.655,A -85,B 0,C 180,E1 -3135.78,E2 -3135.78} C_VEL
LIN {X 0,Y 553.137,Z 597.991,A -85,B 0,C 180,E1 -3137.13,E2 -3137.13} C_VEL
LIN {X 0,Y 553.05,Z 609.553,A -85,B 0,C 180,E1 -3137.407,E2 -3137.407} C_VEL
LIN {X 0,Y 552.864,Z 619.851,A -85,B 0,C 180,E1 -3137.753,E2 -3137.753} C_VEL
LIN {X 0,Y 552.765,Z 629.55,A -85,B 0,C 180,E1 -3138.179,E2 -3138.179} C_VEL
LIN {X 0,Y 552.605,Z 639.09,A -85,B 0,C 180,E1 -3138.701,E2 -3138.701} C_VEL
LIN {X 0,Y 552.443,Z 647.778,A -85,B 0,C 180,E1 -3139.277,E2 -3139.277} C_VEL
LIN {X 0,Y 552.301,Z 655.948,A -85,B 0,C 180,E1 -3139.923,E2 -3139.923} C_VEL
LIN {X 0,Y 552.169,Z 663.833,A -85,B 0,C 180,E1 -3140.661,E2 -3140.661} C_VEL
LIN {X 0,Y 552.045,Z 672.061,A -85,B 0,C 180,E1 -3141.581,E2 -3141.581} C_VEL
LIN {X 0,Y 551.927,Z 678.892,A -85,B 0,C 180,E1 -3142.5,E2 -3142.5} C_VEL
LIN {X 0,Y 551.823,Z 685.847,A -85,B 0,C 180,E1 -3143.64,E2 -3143.64} C_VEL
LIN {X 0,Y 551.723,Z 691.753,A -85,B 0,C 180,E1 -3144.884,E2 -3144.884} C_VEL
LIN {X 0,Y 551.764,Z 695.724,A -85,B 0,C 180,E1 -3145.983,E2 -3145.983} C_VEL
LIN {X 0,Y 551.723,Z 698.672,A -85,B 0,C 180,E1 -3147.079,E2 -3147.079} C_VEL
LIN {X 0,Y 551.657,Z 700.14,A -85,B 0,C 180,E1 -3147.81,E2 -3147.81} C_VEL
LIN {X 0,Y 551.642,Z 701.737,A -85,B 0,C 180,E1 -3149.27,E2 -3149.27} C_VEL
LIN {X 0,Y 551.641,Z 701.996,A -85,B 0,C 180,E1 -3150,E2 -3150} C_VEL
LIN {X 0,Y 551.645,Z 701.213,A -85,B 0,C 180,E1 -3151.46,E2 -3151.46} C_VEL
LIN {X 0,Y 551.657,Z 700.282,A -85,B 0,C 180,E1 -3152.19,E2 -3152.19} C_VEL
LIN {X 0,Y 551.751,Z 697.042,A -85,B 0,C 180,E1 -3153.652,E2 -3153.652} C_VEL
LIN {X 0,Y 551.725,Z 693.491,A -85,B 0,C 180,E1 -3154.75,E2 -3154.75} C_VEL
LIN {X 0,Y 551.836,Z 688.845,A -85,B 0,C 180,E1 -3155.848,E2 -3155.848} C_VEL
LIN {X 0,Y 551.839,Z 682.974,A -85,B 0,C 180,E1 -3156.949,E2 -3156.949} C_VEL
LIN {X 0,Y 551.978,Z 675.682,A -85,B 0,C 180,E1 -3158.051,E2 -3158.051} C_VEL
LIN {X 0,Y 552.123,Z 666.487,A -85,B 0,C 180,E1 -3159.156,E2 -3159.156} C_VEL
LIN {X 0,Y 552.272,Z 658.03,A -85,B 0,C 180,E1 -3159.985,E2 -3159.985} C_VEL
LIN {X 0,Y 552.449,Z 648.995,A -85,B 0,C 180,E1 -3160.723,E2 -3160.723} C_VEL
LIN {X 0,Y 552.59,Z 640.659,A -85,B 0,C 180,E1 -3161.293,E2 -3161.293} C_VEL
LIN {X 0,Y 552.727,Z 631.149,A -85,B 0,C 180,E1 -3161.832,E2 -3161.832} C_VEL
LIN {X 0,Y 552.868,Z 620.929,A -85,B 0,C 180,E1 -3162.294,E2 -3162.294} C_VEL
LIN {X 0,Y 553.009,Z 610.213,A -85,B 0,C 180,E1 -3162.664,E2 -3162.664} C_VEL
LIN {X 0,Y 553.144,Z 599.024,A -85,B 0,C 180,E1 -3162.94,E2 -3162.94} C_VEL
LIN {X 0,Y 553.322,Z 541.861,A -85,B 0,C 180,E1 -3163.707,E2 -3163.707} C_VEL
LIN {X 0,Y 553.319,Z 493.556,A -85,B 0,C 180,E1 -3164.34,E2 -3164.34} C_VEL
LIN {X 0,Y 552.601,Z 488.124,A -85,B 0,C 180,E1 -3164.454,E2 -3164.454} C_VEL
LIN {X 0,Y 552.933,Z 461.31,A -85,B 0,C 180,E1 -3167.582,E2 -3167.582} C_VEL
LIN {X 0,Y 553.37,Z 436.967,A -85,B 0,C 180,E1 -3170.442,E2 -3170.442} C_VEL
LIN {X 0,Y 553.72,Z 413.712,A -85,B 0,C 180,E1 -3173.17,E2 -3173.17} C_VEL
LIN {X 0,Y 554.025,Z 389.729,A -85,B 0,C 180,E1 -3175.993,E2 -3175.993} C_VEL
LIN {X 0,Y 552.945,Z 383.63,A -85,B 0,C 180,E1 -3176.755,E2 -3176.755} C_VEL
LIN {X 0,Y 552.142,Z 379.828,A -85,B 0,C 180,E1 -3177.273,E2 -3177.273} C_VEL
LIN {X 0,Y 552.095,Z 379.711,A -85,B 0,C 180,E1 -3180.61,E2 -3180.61} C_VEL
LIN {X 0,Y 552.115,Z 379.711,A -85,B 0,C 180,E1 -3183.186,E2 -3183.186} C_VEL
LIN {X 0,Y 552.073,Z 379.716,A -85,B 0,C 180,E1 -3185.845,E2 -3185.845} C_VEL
LIN {X 0,Y 552.12,Z 379.708,A -85,B 0,C 180,E1 -3189.061,E2 -3189.061} C_VEL
LIN {X 0,Y 552.071,Z 379.715,A -85,B 0,C 180,E1 -3191.451,E2 -3191.451} C_VEL
LIN {X 0,Y 552.077,Z 379.706,A -85,B 0,C 180,E1 -3194.53,E2 -3194.53} C_VEL
LIN {X 0,Y 552.112,Z 379.715,A -85,B 0,C 180,E1 -3197.587,E2 -3197.587} C_VEL
LIN {X 0,Y 552.129,Z 379.705,A -85,B 0,C 180,E1 -3200.472,E2 -3200.472} C_VEL
LIN {X 0,Y 552.099,Z 379.71,A -85,B 0,C 180,E1 -3203.319,E2 -3203.319} C_VEL
LIN {X 0,Y 552.101,Z 379.711,A -85,B 0,C 180,E1 -3205.937,E2 -3205.937} C_VEL
LIN {X 0,Y 552.124,Z 379.705,A -85,B 0,C 180,E1 -3208.541,E2 -3208.541} C_VEL
LIN {X 0,Y 552.079,Z 379.714,A -85,B 0,C 180,E1 -3211.448,E2 -3211.448} C_VEL
LIN {X 0,Y 552.081,Z 379.711,A -85,B 0,C 180,E1 -3214.353,E2 -3214.353} C_VEL
LIN {X 0,Y 552.096,Z 379.705,A -85,B 0,C 180,E1 -3216.758,E2 -3216.758} C_VEL
LIN {X 0,Y 552.11,Z 379.708,A -85,B 0,C 180,E1 -3219.119,E2 -3219.119} C_VEL
LIN {X 0,Y 552.084,Z 379.714,A -85,B 0,C 180,E1 -3221.443,E2 -3221.443} C_VEL
LIN {X 0,Y 552.093,Z 379.709,A -85,B 0,C 180,E1 -3224.495,E2 -3224.495} C_VEL
LIN {X 0,Y 552.114,Z 379.705,A -85,B 0,C 180,E1 -3226.754,E2 -3226.754} C_VEL
LIN {X 0,Y 552.129,Z 379.7,A -85,B 0,C 180,E1 -3228.993,E2 -3228.993} C_VEL
LIN {X 0,Y 552.114,Z 379.712,A -85,B 0,C 180,E1 -3231.951,E2 -3231.951} C_VEL
LIN {X 0,Y 552.209,Z 379.69,A -85,B 0,C 180,E1 -3234.889,E2 -3234.889} C_VEL
LIN {X 0,Y 552.222,Z 379.702,A -85,B 0,C 180,E1 -3237.812,E2 -3237.812} C_VEL
LIN {X 0,Y 552.226,Z 379.696,A -85,B 0,C 180,E1 -3240,E2 -3240} C_VEL
LIN {X 0,Y 552.178,Z 379.693,A -85,B 0,C 180,E1 -3242.918,E2 -3242.918} C_VEL
LIN {X 0,Y 552.177,Z 379.707,A -85,B 0,C 180,E1 -3245.844,E2 -3245.844} C_VEL
LIN {X 0,Y 552.127,Z 379.701,A -85,B 0,C 180,E1 -3248.786,E2 -3248.786} C_VEL
LIN {X 0,Y 552.106,Z 379.714,A -85,B 0,C 180,E1 -3251.752,E2 -3251.752} C_VEL
LIN {X 0,Y 552.093,Z 379.707,A -85,B 0,C 180,E1 -3254.75,E2 -3254.75} C_VEL
LIN {X 0,Y 552.071,Z 379.717,A -85,B 0,C 180,E1 -3257.79,E2 -3257.79} C_VEL
LIN {X 0,Y 552.055,Z 379.718,A -85,B 0,C 180,E1 -3260.104,E2 -3260.104} C_VEL
LIN {X 0,Y 552.084,Z 379.707,A -85,B 0,C 180,E1 -3262.451,E2 -3262.451} C_VEL
LIN {X 0,Y 552.074,Z 379.712,A -85,B 0,C 180,E1 -3265.331,E2 -3265.331} C_VEL
LIN {X 0,Y 552.049,Z 379.716,A -85,B 0,C 180,E1 -3268.102,E2 -3268.102} C_VEL
LIN {X 0,Y 552.092,Z 379.709,A -85,B 0,C 180,E1 -3270.61,E2 -3270.61} C_VEL
LIN {X 0,Y 552.098,Z 379.709,A -85,B 0,C 180,E1 -3273.187,E2 -3273.187} C_VEL
LIN {X 0,Y 552.068,Z 379.719,A -85,B 0,C 180,E1 -3275.845,E2 -3275.845} C_VEL
LIN {X 0,Y 552.089,Z 379.708,A -85,B 0,C 180,E1 -3278.591,E2 -3278.591} C_VEL
LIN {X 0,Y 552.052,Z 379.708,A -85,B 0,C 180,E1 -3281.452,E2 -3281.452} C_VEL
LIN {X 0,Y 552.069,Z 379.713,A -85,B 0,C 180,E1 -3284.528,E2 -3284.528} C_VEL
LIN {X 0,Y 552.082,Z 379.714,A -85,B 0,C 180,E1 -3287.59,E2 -3287.59} C_VEL
LIN {X 0,Y 552.089,Z 379.708,A -85,B 0,C 180,E1 -3290.943,E2 -3290.943} C_VEL
LIN {X 0,Y 552.048,Z 379.717,A -85,B 0,C 180,E1 -3293.326,E2 -3293.326} C_VEL
LIN {X 0,Y 552.087,Z 379.719,A -85,B 0,C 180,E1 -3295.936,E2 -3295.936} C_VEL
LIN {X 0,Y 552.082,Z 379.714,A -85,B 0,C 180,E1 -3298.538,E2 -3298.538} C_VEL
LIN {X 0,Y 552.07,Z 379.718,A -85,B 0,C 180,E1 -3301.449,E2 -3301.449} C_VEL
LIN {X 0,Y 552.144,Z 379.882,A -85,B 0,C 180,E1 -3302.161,E2 -3302.161} C_VEL
LIN {X 0,Y 554.254,Z 390.012,A -85,B 0,C 180,E1 -3303.45,E2 -3303.45} C_VEL
LIN {X 0,Y 553.87,Z 416.154,A -85,B 0,C 180,E1 -3306.44,E2 -3306.44} C_VEL
LIN {X 0,Y 553.387,Z 443.848,A -85,B 0,C 180,E1 -3309.558,E2 -3309.558} C_VEL
LIN {X 0,Y 553.046,Z 466.221,A -85,B 0,C 180,E1 -3312.051,E2 -3312.051} C_VEL
LIN {X 0,Y 552.695,Z 491.772,A -85,B 0,C 180,E1 -3314.927,E2 -3314.927} C_VEL
LIN {X 0,Y 552.649,Z 497.901,A -85,B 0,C 180,E1 -3315.595,E2 -3315.595} C_VEL
LIN {X 0,Y 553.446,Z 505.493,A -85,B 0,C 180,E1 -3315.733,E2 -3315.733} C_VEL
LIN {X 0,Y 553.128,Z 607.937,A -85,B 0,C 180,E1 -3317.082,E2 -3317.082} C_VEL
LIN {X 0,Y 553.006,Z 620.449,A -85,B 0,C 180,E1 -3317.383,E2 -3317.383} C_VEL
LIN {X 0,Y 552.851,Z 633.365,A -85,B 0,C 180,E1 -3317.845,E2 -3317.845} C_VEL
LIN {X 0,Y 552.69,Z 645.666,A -85,B 0,C 180,E1 -3318.449,E2 -3318.449} C_VEL
LIN {X 0,Y 552.482,Z 657.194,A -85,B 0,C 180,E1 -3319.185,E2 -3319.185} C_VEL
LIN {X 0,Y 552.301,Z 667.602,A -85,B 0,C 180,E1 -3320.016,E2 -3320.016} C_VEL
LIN {X 0,Y 552.126,Z 676.111,A -85,B 0,C 180,E1 -3320.844,E2 -3320.844} C_VEL
LIN {X 0,Y 552.013,Z 683.959,A -85,B 0,C 180,E1 -3321.765,E2 -3321.765} C_VEL
LIN {X 0,Y 551.889,Z 691.621,A -85,B 0,C 180,E1 -3322.868,E2 -3322.868} C_VEL
LIN {X 0,Y 551.867,Z 698.679,A -85,B 0,C 180,E1 -3324.152,E2 -3324.152} C_VEL
LIN {X 0,Y 551.725,Z 703.372,A -85,B 0,C 180,E1 -3325.25,E2 -3325.25} C_VEL
LIN {X 0,Y 551.75,Z 706.958,A -85,B 0,C 180,E1 -3326.348,E2 -3326.348} C_VEL
LIN {X 0,Y 551.723,Z 708.807,A -85,B 0,C 180,E1 -3327.079,E2 -3327.079} C_VEL
LIN {X 0,Y 551.645,Z 711.184,A -85,B 0,C 180,E1 -3328.54,E2 -3328.54} C_VEL
LIN {X 0,Y 551.64,Z 712,A -85,B 0,C 180,E1 -3330,E2 -3330} C_VEL
LIN {X 0,Y 551.645,Z 711.185,A -85,B 0,C 180,E1 -3331.46,E2 -3331.46} C_VEL
LIN {X 0,Y 551.723,Z 708.81,A -85,B 0,C 180,E1 -3332.921,E2 -3332.921} C_VEL
LIN {X 0,Y 551.764,Z 705.896,A -85,B 0,C 180,E1 -3334.017,E2 -3334.017} C_VEL
LIN {X 0,Y 551.723,Z 701.949,A -85,B 0,C 180,E1 -3335.116,E2 -3335.116} C_VEL
LIN {X 0,Y 551.803,Z 696.188,A -85,B 0,C 180,E1 -3336.342,E2 -3336.342} C_VEL
LIN {X 0,Y 551.926,Z 689.237,A -85,B 0,C 180,E1 -3337.5,E2 -3337.5} C_VEL
LIN {X 0,Y 552.082,Z 680.992,A -85,B 0,C 180,E1 -3338.602,E2 -3338.602} C_VEL
LIN {X 0,Y 552.224,Z 672.54,A -85,B 0,C 180,E1 -3339.523,E2 -3339.523} C_VEL
LIN {X 0,Y 552.422,Z 662.095,A -85,B 0,C 180,E1 -3340.445,E2 -3340.445} C_VEL
LIN {X 0,Y 552.621,Z 651.129,A -85,B 0,C 180,E1 -3341.223,E2 -3341.223} C_VEL
LIN {X 0,Y 552.753,Z 640.407,A -85,B 0,C 180,E1 -3341.831,E2 -3341.831} C_VEL
LIN {X 0,Y 552.924,Z 628.764,A -85,B 0,C 180,E1 -3342.339,E2 -3342.339} C_VEL
LIN {X 0,Y 553.058,Z 615.346,A -85,B 0,C 180,E1 -3342.756,E2 -3342.756} C_VEL
LIN {X 0,Y 553.217,Z 602.085,A -85,B 0,C 180,E1 -3343.009,E2 -3343.009} C_VEL
LIN {X 0,Y 553.38,Z 503.72,A -85,B 0,C 180,E1 -3344.292,E2 -3344.292} C_VEL
LIN {X 0,Y 552.651,Z 497.908,A -85,B 0,C 180,E1 -3344.405,E2 -3344.405} C_VEL
LIN {X 0,Y 553.022,Z 469.193,A -85,B 0,C 180,E1 -3347.612,E2 -3347.612} C_VEL
LIN {X 0,Y 553.286,Z 449.217,A -85,B 0,C 180,E1 -3349.836,E2 -3349.836} C_VEL
LIN {X 0,Y 553.598,Z 424.081,A -85,B 0,C 180,E1 -3352.583,E2 -3352.583} C_VEL
LIN {X 0,Y 553.783,Z 402.558,A -85,B 0,C 180,E1 -3354.959,E2 -3354.959} C_VEL
LIN {X 0,Y 553.871,Z 388.215,A -85,B 0,C 180,E1 -3356.567,E2 -3356.567} C_VEL
LIN {X 0,Y 552.08,Z 379.878,A -85,B 0,C 180,E1 -3357.61,E2 -3357.61} C_VEL
LIN {X 0,Y 552.071,Z 379.716,A -85,B 0,C 180,E1 -3360.611,E2 -3360.611} C_VEL
LIN {X 0,Y 552.089,Z 379.712,A -85,B 0,C 180,E1 -3363.188,E2 -3363.188} C_VEL
LIN {X 0,Y 552.066,Z 379.721,A -85,B 0,C 180,E1 -3365.845,E2 -3365.845} C_VEL
LIN {X 0,Y 552.089,Z 379.711,A -85,B 0,C 180,E1 -3368.592,E2 -3368.592} C_VEL
LIN {X 0,Y 552.053,Z 379.718,A -85,B 0,C 180,E1 -3371.452,E2 -3371.452} C_VEL
LIN {X 0,Y 552.076,Z 379.712,A -85,B 0,C 180,E1 -3374.529,E2 -3374.529} C_VEL
LIN {X 0,Y 552.088,Z 379.717,A -85,B 0,C 180,E1 -3377.59,E2 -3377.59} C_VEL
LIN {X 0,Y 552.127,Z 379.705,A -85,B 0,C 180,E1 -3380.472,E2 -3380.472} C_VEL
LIN {X 0,Y 552.098,Z 379.714,A -85,B 0,C 180,E1 -3383.319,E2 -3383.319} C_VEL
LIN {X 0,Y 552.119,Z 379.711,A -85,B 0,C 180,E1 -3385.938,E2 -3385.938} C_VEL
LIN {X 0,Y 552.122,Z 379.706,A -85,B 0,C 180,E1 -3388.541,E2 -3388.541} C_VEL
LIN {X 0,Y 552.1,Z 379.716,A -85,B 0,C 180,E1 -3391.443,E2 -3391.443} C_VEL
LIN {X 0,Y 552.124,Z 379.706,A -85,B 0,C 180,E1 -3394.657,E2 -3394.657} C_VEL
LIN {X 0,Y 552.094,Z 379.717,A -85,B 0,C 180,E1 -3397.549,E2 -3397.549} C_VEL
LIN {X 0,Y 552.148,Z 379.704,A -85,B 0,C 180,E1 -3400.375,E2 -3400.375} C_VEL
LIN {X 0,Y 552.159,Z 379.708,A -85,B 0,C 180,E1 -3402.977,E2 -3402.977} C_VEL
LIN {X 0,Y 552.19,Z 379.898,A -85,B 0,C 180,E1 -3405.964,E2 -3405.964} C_VEL
LIN {X 0,Y 552.423,Z 380.908,A -85,B 0,C 180,E1 -3406.077,E2 -3406.077} C_VEL
LIN {X 0,Y 553.346,Z 384.054,A -85,B 0,C 180,E1 -3406.153,E2 -3406.153} C_VEL
LIN {X 0,Y 553.097,Z 459.965,A -85,B 0,C 180,E1 -3407.175,E2 -3407.175} C_VEL
LIN {X 0,Y 553.029,Z 473.226,A -85,B 0,C 180,E1 -3407.5,E2 -3407.5} C_VEL
LIN {X 0,Y 552.856,Z 486.349,A -85,B 0,C 180,E1 -3407.995,E2 -3407.995} C_VEL
LIN {X 0,Y 552.747,Z 496.656,A -85,B 0,C 180,E1 -3408.515,E2 -3408.515} C_VEL
LIN {X 0,Y 552.574,Z 505.935,A -85,B 0,C 180,E1 -3409.094,E2 -3409.094} C_VEL
LIN {X 0,Y 552.398,Z 514.483,A -85,B 0,C 180,E1 -3409.74,E2 -3409.74} C_VEL
LIN {X 0,Y 552.283,Z 522.635,A -85,B 0,C 180,E1 -3410.478,E2 -3410.478} C_VEL
LIN {X 0,Y 552.15,Z 529.534,A -85,B 0,C 180,E1 -3411.214,E2 -3411.214} C_VEL
LIN {X 0,Y 551.994,Z 536.746,A -85,B 0,C 180,E1 -3412.133,E2 -3412.133} C_VEL
LIN {X 0,Y 551.888,Z 542.955,A -85,B 0,C 180,E1 -3413.088,E2 -3413.088} C_VEL
LIN {X 0,Y 551.869,Z 547.374,A -85,B 0,C 180,E1 -3413.897,E2 -3413.897} C_VEL
LIN {X 0,Y 551.723,Z 551.843,A -85,B 0,C 180,E1 -3414.884,E2 -3414.884} C_VEL
LIN {X 0,Y 551.764,Z 555.756,A -85,B 0,C 180,E1 -3415.983,E2 -3415.983} C_VEL
LIN {X 0,Y 551.723,Z 558.704,A -85,B 0,C 180,E1 -3417.079,E2 -3417.079} C_VEL
LIN {X 0,Y 551.656,Z 560.135,A -85,B 0,C 180,E1 -3417.81,E2 -3417.81} C_VEL
LIN {X 0,Y 551.642,Z 561.733,A -85,B 0,C 180,E1 -3419.27,E2 -3419.27} C_VEL
LIN {X 0,Y 551.641,Z 561.996,A -85,B 0,C 180,E1 -3420,E2 -3420} C_VEL
LIN {X 0,Y 551.645,Z 561.215,A -85,B 0,C 180,E1 -3421.46,E2 -3421.46} C_VEL
LIN {X 0,Y 551.657,Z 560.28,A -85,B 0,C 180,E1 -3422.19,E2 -3422.19} C_VEL
LIN {X 0,Y 551.751,Z 557.072,A -85,B 0,C 180,E1 -3423.652,E2 -3423.652} C_VEL
LIN {X 0,Y 551.729,Z 553.599,A -85,B 0,C 180,E1 -3424.749,E2 -3424.749} C_VEL
LIN {X 0,Y 551.859,Z 548.974,A -85,B 0,C 180,E1 -3425.848,E2 -3425.848} C_VEL
LIN {X 0,Y 551.863,Z 544.274,A -85,B 0,C 180,E1 -3426.765,E2 -3426.765} C_VEL
LIN {X 0,Y 551.949,Z 538.586,A -85,B 0,C 180,E1 -3427.683,E2 -3427.683} C_VEL
LIN {X 0,Y 552.101,Z 531.717,A -85,B 0,C 180,E1 -3428.602,E2 -3428.602} C_VEL
LIN {X 0,Y 552.202,Z 525.237,A -85,B 0,C 180,E1 -3429.339,E2 -3429.339} C_VEL
LIN {X 0,Y 552.325,Z 516.493,A -85,B 0,C 180,E1 -3430.169,E2 -3430.169} C_VEL
LIN {X 0,Y 552.502,Z 508.356,A -85,B 0,C 180,E1 -3430.814,E2 -3430.814} C_VEL
LIN {X 0,Y 552.678,Z 499.088,A -85,B 0,C 180,E1 -3431.425,E2 -3431.425} C_VEL
LIN {X 0,Y 552.786,Z 490.622,A -85,B 0,C 180,E1 -3431.888,E2 -3431.888} C_VEL
LIN {X 0,Y 552.92,Z 480.642,A -85,B 0,C 180,E1 -3432.325,E2 -3432.325} C_VEL
LIN {X 0,Y 553.055,Z 469.716,A -85,B 0,C 180,E1 -3432.686,E2 -3432.686} C_VEL
LIN {X 0,Y 553.122,Z 458.563,A -85,B 0,C 180,E1 -3432.941,E2 -3432.941} C_VEL
LIN {X 0,Y 553.226,Z 383.407,A -85,B 0,C 180,E1 -3433.95,E2 -3433.95} C_VEL
LIN {X 0,Y 552.283,Z 380.363,A -85,B 0,C 180,E1 -3434.054,E2 -3434.054} C_VEL
LIN {X 0,Y 552.173,Z 379.713,A -85,B 0,C 180,E1 -3434.244,E2 -3434.244} C_VEL
LIN {X 0,Y 552.119,Z 379.71,A -85,B 0,C 180,E1 -3437.314,E2 -3437.314} C_VEL
LIN {X 0,Y 552.13,Z 379.706,A -85,B 0,C 180,E1 -3440.101,E2 -3440.101} C_VEL
LIN {X 0,Y 552.085,Z 379.712,A -85,B 0,C 180,E1 -3442.921,E2 -3442.921} C_VEL
LIN {X 0,Y 551.438,Z 379.794,A -85,B 0,C 180,E1 -3443.53,E2 -3443.53} C_VEL
LIN {X 0,Y 548.605,Z 380.149,A -85,B 0,C 180,E1 -3444.519,E2 -3444.519} C_VEL
LIN {X 0,Y 546.198,Z 380.446,A -85,B 0,C 180,E1 -3445.314,E2 -3445.314} C_VEL
LIN {X 0,Y 545.159,Z 380.573,A -85,B 0,C 180,E1 -3445.929,E2 -3445.929} C_VEL
LIN {X 0,Y 545.072,Z 380.584,A -85,B 0,C 180,E1 -3446.137,E2 -3446.137} C_VEL
LIN {X 0,Y 545.062,Z 380.584,A -85,B 0,C 180,E1 -3449.339,E2 -3449.339} C_VEL
LIN {X 0,Y 545.058,Z 380.586,A -85,B 0,C 180,E1 -3451.915,E2 -3451.915} C_VEL
LIN {X 0,Y 545.062,Z 380.588,A -85,B 0,C 180,E1 -3454.565,E2 -3454.565} C_VEL
LIN {X 0,Y 545.034,Z 380.588,A -85,B 0,C 180,E1 -3457.304,E2 -3457.304} C_VEL
LIN {X 0,Y 545.067,Z 380.586,A -85,B 0,C 180,E1 -3460.143,E2 -3460.143} C_VEL
LIN {X 0,Y 545.041,Z 380.595,A -85,B 0,C 180,E1 -3462.694,E2 -3462.694} C_VEL
LIN {X 0,Y 545.032,Z 380.59,A -85,B 0,C 180,E1 -3465.171,E2 -3465.171} C_VEL
LIN {X 0,Y 545.067,Z 380.584,A -85,B 0,C 180,E1 -3467.896,E2 -3467.896} C_VEL
LIN {X 0,Y 545.08,Z 380.583,A -85,B 0,C 180,E1 -3470.818,E2 -3470.818} C_VEL
LIN {X 0,Y 545.036,Z 380.589,A -85,B 0,C 180,E1 -3473.619,E2 -3473.619} C_VEL
LIN {X 0,Y 545.068,Z 380.59,A -85,B 0,C 180,E1 -3476.328,E2 -3476.328} C_VEL
LIN {X 0,Y 545.067,Z 380.588,A -85,B 0,C 180,E1 -3478.952,E2 -3478.952} C_VEL
LIN {X 0,Y 545.078,Z 380.585,A -85,B 0,C 180,E1 -3481.506,E2 -3481.506} C_VEL
LIN {X 0,Y 545.123,Z 380.778,A -85,B 0,C 180,E1 -3482.64,E2 -3482.64} C_VEL
LIN {X 0,Y 547.14,Z 390.401,A -85,B 0,C 180,E1 -3483.9,E2 -3483.9} C_VEL
LIN {X 0,Y 546.805,Z 414.132,A -85,B 0,C 180,E1 -3486.72,E2 -3486.72} C_VEL
LIN {X 0,Y 546.406,Z 439.17,A -85,B 0,C 180,E1 -3489.679,E2 -3489.679} C_VEL
LIN {X 0,Y 545.906,Z 465.432,A -85,B 0,C 180,E1 -3492.776,E2 -3492.776} C_VEL
LIN {X 0,Y 545.633,Z 488.011,A -85,B 0,C 180,E1 -3495.435,E2 -3495.435} C_VEL
LIN {X 0,Y 546.17,Z 492.46,A -85,B 0,C 180,E1 -3495.544,E2 -3495.544} C_VEL
LIN {X 0,Y 546.535,Z 497.743,A -85,B 0,C 180,E1 -3495.624,E2 -3495.624} C_VEL
LIN {X 0,Y 546.238,Z 598.016,A -85,B 0,C 180,E1 -3496.964,E2 -3496.964} C_VEL
LIN {X 0,Y 546.127,Z 609.549,A -85,B 0,C 180,E1 -3497.245,E2 -3497.245} C_VEL
LIN {X 0,Y 545.937,Z 619.838,A -85,B 0,C 180,E1 -3497.595,E2 -3497.595} C_VEL
LIN {X 0,Y 545.817,Z 629.355,A -85,B 0,C 180,E1 -3498.017,E2 -3498.017} C_VEL
LIN {X 0,Y 545.683,Z 637.563,A -85,B 0,C 180,E1 -3498.461,E2 -3498.461} C_VEL
LIN {X 0,Y 545.534,Z 646.518,A -85,B 0,C 180,E1 -3499.046,E2 -3499.046} C_VEL
LIN {X 0,Y 545.293,Z 655.946,A -85,B 0,C 180,E1 -3499.792,E2 -3499.792} C_VEL
LIN {X 0,Y 545.156,Z 663.83,A -85,B 0,C 180,E1 -3500.539,E2 -3500.539} C_VEL
LIN {X 0,Y 545.037,Z 670.547,A -85,B 0,C 180,E1 -3501.286,E2 -3501.286} C_VEL
LIN {X 0,Y 544.896,Z 677.616,A -85,B 0,C 180,E1 -3502.217,E2 -3502.217} C_VEL
LIN {X 0,Y 544.796,Z 683.511,A -85,B 0,C 180,E1 -3503.147,E2 -3503.147} C_VEL
LIN {X 0,Y 544.778,Z 688.414,A -85,B 0,C 180,E1 -3504.076,E2 -3504.076} C_VEL
LIN {X 0,Y 544.628,Z 693.146,A -85,B 0,C 180,E1 -3505.189,E2 -3505.189} C_VEL
LIN {X 0,Y 544.669,Z 696.779,A -85,B 0,C 180,E1 -3506.301,E2 -3506.301} C_VEL
LIN {X 0,Y 544.65,Z 698.667,A -85,B 0,C 180,E1 -3507.041,E2 -3507.041} C_VEL
LIN {X 0,Y 544.571,Z 700.14,A -85,B 0,C 180,E1 -3507.781,E2 -3507.781} C_VEL
LIN {X 0,Y 544.542,Z 701.73,A -85,B 0,C 180,E1 -3509.261,E2 -3509.261} C_VEL
LIN {X 0,Y 544.542,Z 701.996,A -85,B 0,C 180,E1 -3510,E2 -3510} C_VEL
LIN {X 0,Y 544.546,Z 701.206,A -85,B 0,C 180,E1 -3511.479,E2 -3511.479} C_VEL
LIN {X 0,Y 544.572,Z 700.283,A -85,B 0,C 180,E1 -3512.219,E2 -3512.219} C_VEL
LIN {X 0,Y 544.669,Z 697.035,A -85,B 0,C 180,E1 -3513.699,E2 -3513.699} C_VEL
LIN {X 0,Y 544.628,Z 693.482,A -85,B 0,C 180,E1 -3514.812,E2 -3514.812} C_VEL
LIN {X 0,Y 544.753,Z 688.834,A -85,B 0,C 180,E1 -3515.924,E2 -3515.924} C_VEL
LIN {X 0,Y 544.782,Z 682.962,A -85,B 0,C 180,E1 -3517.04,E2 -3517.04} C_VEL
LIN {X 0,Y 544.91,Z 675.678,A -85,B 0,C 180,E1 -3518.156,E2 -3518.156} C_VEL
LIN {X 0,Y 545.077,Z 666.473,A -85,B 0,C 180,E1 -3519.275,E2 -3519.275} C_VEL
LIN {X 0,Y 545.24,Z 658.014,A -85,B 0,C 180,E1 -3520.115,E2 -3520.115} C_VEL
LIN {X 0,Y 545.465,Z 648.975,A -85,B 0,C 180,E1 -3520.862,E2 -3520.862} C_VEL
LIN {X 0,Y 545.642,Z 639.401,A -85,B 0,C 180,E1 -3521.516,E2 -3521.516} C_VEL
LIN {X 0,Y 545.77,Z 631.118,A -85,B 0,C 180,E1 -3521.985,E2 -3521.985} C_VEL
LIN {X 0,Y 545.937,Z 620.893,A -85,B 0,C 180,E1 -3522.453,E2 -3522.453} C_VEL
LIN {X 0,Y 546.075,Z 610.945,A -85,B 0,C 180,E1 -3522.804,E2 -3522.804} C_VEL
LIN {X 0,Y 546.237,Z 600.207,A -85,B 0,C 180,E1 -3523.083,E2 -3523.083} C_VEL
LIN {X 0,Y 546.346,Z 575.807,A -85,B 0,C 180,E1 -3523.436,E2 -3523.436} C_VEL
LIN {X 0,Y 546.405,Z 494.118,A -85,B 0,C 180,E1 -3524.518,E2 -3524.518} C_VEL
LIN {X 0,Y 545.631,Z 488.28,A -85,B 0,C 180,E1 -3524.632,E2 -3524.632} C_VEL
LIN {X 0,Y 545.975,Z 461.977,A -85,B 0,C 180,E1 -3527.719,E2 -3527.719} C_VEL
LIN {X 0,Y 546.431,Z 436.633,A -85,B 0,C 180,E1 -3530.714,E2 -3530.714} C_VEL
LIN {X 0,Y 546.81,Z 414.917,A -85,B 0,C 180,E1 -3533.28,E2 -3533.28} C_VEL
LIN {X 0,Y 547.151,Z 391.35,A -85,B 0,C 180,E1 -3536.079,E2 -3536.079} C_VEL
LIN {X 0,Y 546.634,Z 387.703,A -85,B 0,C 180,E1 -3536.537,E2 -3536.537} C_VEL
LIN {X 0,Y 545.095,Z 380.772,A -85,B 0,C 180,E1 -3537.455,E2 -3537.455} C_VEL
LIN {X 0,Y 545.047,Z 380.591,A -85,B 0,C 180,E1 -3540.24,E2 -3540.24} C_VEL
LIN {X 0,Y 545.079,Z 380.586,A -85,B 0,C 180,E1 -3543.062,E2 -3543.062} C_VEL
LIN {X 0,Y 545.023,Z 380.597,A -85,B 0,C 180,E1 -3545.671,E2 -3545.671} C_VEL
LIN {X 0,Y 545.048,Z 380.589,A -85,B 0,C 180,E1 -3548.238,E2 -3548.238} C_VEL
LIN {X 0,Y 545.07,Z 380.581,A -85,B 0,C 180,E1 -3550.471,E2 -3550.471} C_VEL
LIN {X 0,Y 545.019,Z 380.593,A -85,B 0,C 180,E1 -3553.113,E2 -3553.113} C_VEL
LIN {X 0,Y 545.049,Z 380.588,A -85,B 0,C 180,E1 -3556.227,E2 -3556.227} C_VEL
LIN {X 0,Y 545.023,Z 380.59,A -85,B 0,C 180,E1 -3558.88,E2 -3558.88} C_VEL
LIN {X 0,Y 545.048,Z 380.593,A -85,B 0,C 180,E1 -3561.762,E2 -3561.762} C_VEL
LIN {X 0,Y 545.026,Z 380.589,A -85,B 0,C 180,E1 -3564.531,E2 -3564.531} C_VEL
LIN {X 0,Y 545.067,Z 380.583,A -85,B 0,C 180,E1 -3567.211,E2 -3567.211} C_VEL
LIN {X 0,Y 545.066,Z 380.59,A -85,B 0,C 180,E1 -3569.81,E2 -3569.81} C_VEL
LIN {X 0,Y 545.027,Z 380.589,A -85,B 0,C 180,E1 -3572.841,E2 -3572.841} C_VEL
LIN {X 0,Y 545.029,Z 380.596,A -85,B 0,C 180,E1 -3575.63,E2 -3575.63} C_VEL
LIN {X 0,Y 545.069,Z 380.586,A -85,B 0,C 180,E1 -3578.18,E2 -3578.18} C_VEL
LIN {X 0,Y 545.108,Z 380.579,A -85,B 0,C 180,E1 -3580.414,E2 -3580.414} C_VEL
LIN {X 0,Y 545.028,Z 380.591,A -85,B 0,C 180,E1 -3583.52,E2 -3583.52} C_VEL
LIN {X 0,Y 545.085,Z 380.589,A -85,B 0,C 180,E1 -3585.82,E2 -3585.82} C_VEL
LIN {X 0,Y 545.075,Z 380.577,A -85,B 0,C 180,E1 -3588.848,E2 -3588.848} C_VEL
LIN {X 0,Y 545.072,Z 380.591,A -85,B 0,C 180,E1 -3591.846,E2 -3591.846} C_VEL
LIN {X 0,Y 545.167,Z 380.567,A -85,B 0,C 180,E1 -3594.823,E2 -3594.823} C_VEL
LIN {X 0,Y 545.193,Z 380.576,A -85,B 0,C 180,E1 -3597.784,E2 -3597.784} C_VEL
LIN {X 0,Y 545.194,Z 380.572,A -85,B 0,C 180,E1 -3600,E2 -3600} C_VEL
LIN {X 0,Y 545.146,Z 380.569,A -85,B 0,C 180,E1 -3602.956,E2 -3602.956} C_VEL
LIN {X 0,Y 545.128,Z 380.584,A -85,B 0,C 180,E1 -3605.92,E2 -3605.92} C_VEL
LIN {X 0,Y 545.071,Z 380.58,A -85,B 0,C 180,E1 -3608.901,E2 -3608.901} C_VEL
LIN {X 0,Y 545.07,Z 380.591,A -85,B 0,C 180,E1 -3611.906,E2 -3611.906} C_VEL
LIN {X 0,Y 545.042,Z 380.586,A -85,B 0,C 180,E1 -3614.945,E2 -3614.945} C_VEL
LIN {X 0,Y 545.037,Z 380.593,A -85,B 0,C 180,E1 -3618.027,E2 -3618.027} C_VEL
LIN {X 0,Y 545.01,Z 380.592,A -85,B 0,C 180,E1 -3620.375,E2 -3620.375} C_VEL
LIN {X 0,Y 545.03,Z 380.584,A -85,B 0,C 180,E1 -3622.758,E2 -3622.758} C_VEL
LIN {X 0,Y 545.026,Z 380.592,A -85,B 0,C 180,E1 -3625.492,E2 -3625.492} C_VEL
LIN {X 0,Y 545.034,Z 380.585,A -85,B 0,C 180,E1 -3628.496,E2 -3628.496} C_VEL
LIN {X 0,Y 545.056,Z 380.585,A -85,B 0,C 180,E1 -3631.049,E2 -3631.049} C_VEL
LIN {X 0,Y 545.044,Z 380.593,A -85,B 0,C 180,E1 -3633.673,E2 -3633.673} C_VEL
LIN {X 0,Y 545.004,Z 380.594,A -85,B 0,C 180,E1 -3636.383,E2 -3636.383} C_VEL
LIN {X 0,Y 545.034,Z 380.588,A -85,B 0,C 180,E1 -3639.314,E2 -3639.314} C_VEL
LIN {X 0,Y 545.03,Z 380.588,A -85,B 0,C 180,E1 -3642.108,E2 -3642.108} C_VEL
LIN {X 0,Y 545.019,Z 380.591,A -85,B 0,C 180,E1 -3645.172,E2 -3645.172} C_VEL
LIN {X 0,Y 545.031,Z 380.589,A -85,B 0,C 180,E1 -3647.892,E2 -3647.892} C_VEL
LIN {X 0,Y 545.044,Z 380.586,A -85,B 0,C 180,E1 -3650.815,E2 -3650.815} C_VEL
LIN {X 0,Y 545,Z 380.598,A -85,B 0,C 180,E1 -3653.616,E2 -3653.616} C_VEL
LIN {X 0,Y 545.036,Z 380.593,A -85,B 0,C 180,E1 -3656.326,E2 -3656.326} C_VEL
LIN {X 0,Y 545.035,Z 380.591,A -85,B 0,C 180,E1 -3658.95,E2 -3658.95} C_VEL
LIN {X 0,Y 545.067,Z 380.766,A -85,B 0,C 180,E1 -3661.951,E2 -3661.951} C_VEL
LIN {X 0,Y 547.338,Z 391.089,A -85,B 0,C 180,E1 -3663.294,E2 -3663.294} C_VEL
LIN {X 0,Y 547.008,Z 413.86,A -85,B 0,C 180,E1 -3665.937,E2 -3665.937} C_VEL
LIN {X 0,Y 546.513,Z 441.358,A -85,B 0,C 180,E1 -3669.092,E2 -3669.092} C_VEL
LIN {X 0,Y 546.041,Z 467.463,A -85,B 0,C 180,E1 -3672.007,E2 -3672.007} C_VEL
LIN {X 0,Y 545.762,Z 489.757,A -85,B 0,C 180,E1 -3674.502,E2 -3674.502} C_VEL
LIN {X 0,Y 545.692,Z 498.166,A -85,B 0,C 180,E1 -3675.42,E2 -3675.42} C_VEL
LIN {X 0,Y 546.577,Z 505.561,A -85,B 0,C 180,E1 -3675.551,E2 -3675.551} C_VEL
LIN {X 0,Y 546.224,Z 607.937,A -85,B 0,C 180,E1 -3676.916,E2 -3676.916} C_VEL
LIN {X 0,Y 546.086,Z 621.211,A -85,B 0,C 180,E1 -3677.244,E2 -3677.244} C_VEL
LIN {X 0,Y 545.895,Z 633.365,A -85,B 0,C 180,E1 -3677.688,E2 -3677.688} C_VEL
LIN {X 0,Y 545.731,Z 645.665,A -85,B 0,C 180,E1 -3678.3,E2 -3678.3} C_VEL
LIN {X 0,Y 545.495,Z 657.192,A -85,B 0,C 180,E1 -3679.045,E2 -3679.045} C_VEL
LIN {X 0,Y 545.29,Z 667.603,A -85,B 0,C 180,E1 -3679.886,E2 -3679.886} C_VEL
LIN {X 0,Y 545.085,Z 676.111,A -85,B 0,C 180,E1 -3680.725,E2 -3680.725} C_VEL
LIN {X 0,Y 544.978,Z 683.959,A -85,B 0,C 180,E1 -3681.658,E2 -3681.658} C_VEL
LIN {X 0,Y 544.824,Z 691.621,A -85,B 0,C 180,E1 -3682.775,E2 -3682.775} C_VEL
LIN {X 0,Y 544.776,Z 698.679,A -85,B 0,C 180,E1 -3684.076,E2 -3684.076} C_VEL
LIN {X 0,Y 544.628,Z 703.372,A -85,B 0,C 180,E1 -3685.188,E2 -3685.188} C_VEL
LIN {X 0,Y 544.669,Z 706.958,A -85,B 0,C 180,E1 -3686.301,E2 -3686.301} C_VEL
LIN {X 0,Y 544.65,Z 708.807,A -85,B 0,C 180,E1 -3687.041,E2 -3687.041} C_VEL
LIN {X 0,Y 544.546,Z 711.183,A -85,B 0,C 180,E1 -3688.521,E2 -3688.521} C_VEL
LIN {X 0,Y 544.541,Z 712,A -85,B 0,C 180,E1 -3690,E2 -3690} C_VEL
LIN {X 0,Y 544.546,Z 711.185,A -85,B 0,C 180,E1 -3691.479,E2 -3691.479} C_VEL
LIN {X 0,Y 544.65,Z 708.81,A -85,B 0,C 180,E1 -3692.959,E2 -3692.959} C_VEL
LIN {X 0,Y 544.684,Z 705.896,A -85,B 0,C 180,E1 -3694.069,E2 -3694.069} C_VEL
LIN {X 0,Y 544.653,Z 701.948,A -85,B 0,C 180,E1 -3695.182,E2 -3695.182} C_VEL
LIN {X 0,Y 544.74,Z 696.703,A -85,B 0,C 180,E1 -3696.328,E2 -3696.328} C_VEL
LIN {X 0,Y 544.836,Z 690.467,A -85,B 0,C 180,E1 -3697.411,E2 -3697.411} C_VEL
LIN {X 0,Y 545.007,Z 682.478,A -85,B 0,C 180,E1 -3698.528,E2 -3698.528} C_VEL
LIN {X 0,Y 545.154,Z 674.334,A -85,B 0,C 180,E1 -3699.461,E2 -3699.461} C_VEL
LIN {X 0,Y 545.368,Z 664.398,A -85,B 0,C 180,E1 -3700.394,E2 -3700.394} C_VEL
LIN {X 0,Y 545.576,Z 653.539,A -85,B 0,C 180,E1 -3701.211,E2 -3701.211} C_VEL
LIN {X 0,Y 545.763,Z 642.172,A -85,B 0,C 180,E1 -3701.89,E2 -3701.89} C_VEL
LIN {X 0,Y 545.932,Z 629.973,A -85,B 0,C 180,E1 -3702.452,E2 -3702.452} C_VEL
LIN {X 0,Y 546.121,Z 617.174,A -85,B 0,C 180,E1 -3702.873,E2 -3702.873} C_VEL
LIN {X 0,Y 546.299,Z 603.6,A -85,B 0,C 180,E1 -3703.153,E2 -3703.153} C_VEL
LIN {X 0,Y 546.394,Z 503.753,A -85,B 0,C 180,E1 -3704.478,E2 -3704.478} C_VEL
LIN {X 0,Y 545.664,Z 497.925,A -85,B 0,C 180,E1 -3704.593,E2 -3704.593} C_VEL
LIN {X 0,Y 546.01,Z 471.988,A -85,B 0,C 180,E1 -3707.48,E2 -3707.48} C_VEL
LIN {X 0,Y 546.365,Z 444.174,A -85,B 0,C 180,E1 -3710.519,E2 -3710.519} C_VEL
LIN {X 0,Y 546.683,Z 417.543,A -85,B 0,C 180,E1 -3713.486,E2 -3713.486} C_VEL
LIN {X 0,Y 546.992,Z 392.478,A -85,B 0,C 180,E1 -3716.313,E2 -3716.313} C_VEL
LIN {X 0,Y 546.508,Z 387.525,A -85,B 0,C 180,E1 -3716.902,E2 -3716.902} C_VEL
LIN {X 0,Y 545.036,Z 380.718,A -85,B 0,C 180,E1 -3717.789,E2 -3717.789} C_VEL
LIN {X 0,Y 545.022,Z 380.598,A -85,B 0,C 180,E1 -3720.236,E2 -3720.236} C_VEL
LIN {X 0,Y 545.058,Z 380.587,A -85,B 0,C 180,E1 -3723.058,E2 -3723.058} C_VEL
LIN {X 0,Y 545.016,Z 380.598,A -85,B 0,C 180,E1 -3725.67,E2 -3725.67} C_VEL
LIN {X 0,Y 545.03,Z 380.594,A -85,B 0,C 180,E1 -3728.239,E2 -3728.239} C_VEL
LIN {X 0,Y 544.996,Z 380.594,A -85,B 0,C 180,E1 -3731.123,E2 -3731.123} C_VEL
LIN {X 0,Y 545.031,Z 380.594,A -85,B 0,C 180,E1 -3734.132,E2 -3734.132} C_VEL
LIN {X 0,Y 545.019,Z 380.59,A -85,B 0,C 180,E1 -3736.887,E2 -3736.887} C_VEL
LIN {X 0,Y 545.059,Z 380.592,A -85,B 0,C 180,E1 -3739.857,E2 -3739.857} C_VEL
LIN {X 0,Y 545.028,Z 380.59,A -85,B 0,C 180,E1 -3742.695,E2 -3742.695} C_VEL
LIN {X 0,Y 545.07,Z 380.592,A -85,B 0,C 180,E1 -3745.609,E2 -3745.609} C_VEL
LIN {X 0,Y 545.06,Z 380.586,A -85,B 0,C 180,E1 -3748.321,E2 -3748.321} C_VEL
LIN {X 0,Y 545.071,Z 380.59,A -85,B 0,C 180,E1 -3751.256,E2 -3751.256} C_VEL
LIN {X 0,Y 545.072,Z 380.584,A -85,B 0,C 180,E1 -3754.497,E2 -3754.497} C_VEL
LIN {X 0,Y 545.039,Z 380.596,A -85,B 0,C 180,E1 -3757.242,E2 -3757.242} C_VEL
LIN {X 0,Y 545.12,Z 380.58,A -85,B 0,C 180,E1 -3760.415,E2 -3760.415} C_VEL
LIN {X 0,Y 545.075,Z 380.592,A -85,B 0,C 180,E1 -3763.521,E2 -3763.521} C_VEL
LIN {X 0,Y 545.147,Z 380.753,A -85,B 0,C 180,E1 -3765.785,E2 -3765.785} C_VEL
LIN {X 0,Y 545.383,Z 381.761,A -85,B 0,C 180,E1 -3765.904,E2 -3765.904} C_VEL
LIN {X 0,Y 546.486,Z 385.805,A -85,B 0,C 180,E1 -3765.999,E2 -3765.999} C_VEL
LIN {X 0,Y 546.205,Z 461.131,A -85,B 0,C 180,E1 -3767.034,E2 -3767.034} C_VEL
LIN {X 0,Y 546.115,Z 474.276,A -85,B 0,C 180,E1 -3767.363,E2 -3767.363} C_VEL
LIN {X 0,Y 545.949,Z 487.372,A -85,B 0,C 180,E1 -3767.859,E2 -3767.859} C_VEL
LIN {X 0,Y 545.773,Z 498.804,A -85,B 0,C 180,E1 -3768.45,E2 -3768.45} C_VEL
LIN {X 0,Y 545.599,Z 509.354,A -85,B 0,C 180,E1 -3769.141,E2 -3769.141} C_VEL
LIN {X 0,Y 545.398,Z 519.665,A -85,B 0,C 180,E1 -3769.982,E2 -3769.982} C_VEL
LIN {X 0,Y 545.222,Z 528.894,A -85,B 0,C 180,E1 -3770.915,E2 -3770.915} C_VEL
LIN {X 0,Y 545.036,Z 537.719,A -85,B 0,C 180,E1 -3772.032,E2 -3772.032} C_VEL
LIN {X 0,Y 544.919,Z 543.948,A -85,B 0,C 180,E1 -3772.999,E2 -3772.999} C_VEL
LIN {X 0,Y 544.885,Z 549.593,A -85,B 0,C 180,E1 -3774.077,E2 -3774.077} C_VEL
LIN {X 0,Y 544.737,Z 554.242,A -85,B 0,C 180,E1 -3775.19,E2 -3775.19} C_VEL
LIN {X 0,Y 544.733,Z 557.843,A -85,B 0,C 180,E1 -3776.301,E2 -3776.301} C_VEL
LIN {X 0,Y 544.623,Z 561.06,A -85,B 0,C 180,E1 -3777.781,E2 -3777.781} C_VEL
LIN {X 0,Y 544.609,Z 562.587,A -85,B 0,C 180,E1 -3779.261,E2 -3779.261} C_VEL
LIN {X 0,Y 544.605,Z 562.852,A -85,B 0,C 180,E1 -3780,E2 -3780} C_VEL
LIN {X 0,Y 544.622,Z 562.056,A -85,B 0,C 180,E1 -3781.479,E2 -3781.479} C_VEL
LIN {X 0,Y 544.617,Z 561.154,A -85,B 0,C 180,E1 -3782.219,E2 -3782.219} C_VEL
LIN {X 0,Y 544.694,Z 559.784,A -85,B 0,C 180,E1 -3782.958,E2 -3782.958} C_VEL
LIN {X 0,Y 544.755,Z 555.803,A -85,B 0,C 180,E1 -3784.44,E2 -3784.44} C_VEL
LIN {X 0,Y 544.806,Z 551.601,A -85,B 0,C 180,E1 -3785.552,E2 -3785.552} C_VEL
LIN {X 0,Y 544.842,Z 546.219,A -85,B 0,C 180,E1 -3786.667,E2 -3786.667} C_VEL
LIN {X 0,Y 544.969,Z 539.423,A -85,B 0,C 180,E1 -3787.782,E2 -3787.782} C_VEL
LIN {X 0,Y 545.143,Z 532.515,A -85,B 0,C 180,E1 -3788.713,E2 -3788.713} C_VEL
LIN {X 0,Y 545.236,Z 525.993,A -85,B 0,C 180,E1 -3789.459,E2 -3789.459} C_VEL
LIN {X 0,Y 545.392,Z 517.198,A -85,B 0,C 180,E1 -3790.3,E2 -3790.3} C_VEL
LIN {X 0,Y 545.592,Z 507.692,A -85,B 0,C 180,E1 -3791.047,E2 -3791.047} C_VEL
LIN {X 0,Y 545.806,Z 497.898,A -85,B 0,C 180,E1 -3791.675,E2 -3791.675} C_VEL
LIN {X 0,Y 545.959,Z 486.39,A -85,B 0,C 180,E1 -3792.263,E2 -3792.263} C_VEL
LIN {X 0,Y 546.128,Z 472.493,A -85,B 0,C 180,E1 -3792.779,E2 -3792.779} C_VEL
LIN {X 0,Y 546.214,Z 459.723,A -85,B 0,C 180,E1 -3793.084,E2 -3793.084} C_VEL
LIN {X 0,Y 546.338,Z 384.777,A -85,B 0,C 180,E1 -3794.11,E2 -3794.11} C_VEL
LIN {X 0,Y 545.272,Z 381.415,A -85,B 0,C 180,E1 -3794.211,E2 -3794.211} C_VEL
LIN {X 0,Y 545.166,Z 380.641,A -85,B 0,C 180,E1 -3794.358,E2 -3794.358} C_VEL
LIN {X 0,Y 545.08,Z 380.587,A -85,B 0,C 180,E1 -3797.422,E2 -3797.422} C_VEL
LIN {X 0,Y 545.096,Z 380.585,A -85,B 0,C 180,E1 -3800.372,E2 -3800.372} C_VEL
LIN {X 0,Y 545.082,Z 380.583,A -85,B 0,C 180,E1 -3803.559,E2 -3803.559} C_VEL
LIN {X 0,Y 545.072,Z 380.584,A -85,B 0,C 180,E1 -3806.137,E2 -3806.137} C_VEL
LIN {X 0,Y 544.398,Z 380.676,A -85,B 0,C 180,E1 -3806.753,E2 -3806.753} C_VEL
LIN {X 0,Y 541.539,Z 381.028,A -85,B 0,C 180,E1 -3807.754,E2 -3807.754} C_VEL
LIN {X 0,Y 539.127,Z 381.328,A -85,B 0,C 180,E1 -3808.56,E2 -3808.56} C_VEL
LIN {X 0,Y 538.094,Z 381.454,A -85,B 0,C 180,E1 -3809.182,E2 -3809.182} C_VEL
LIN {X 0,Y 538.01,Z 381.462,A -85,B 0,C 180,E1 -3809.392,E2 -3809.392} C_VEL
LIN {X 0,Y 538.02,Z 381.466,A -85,B 0,C 180,E1 -3812.383,E2 -3812.383} C_VEL
LIN {X 0,Y 537.997,Z 381.469,A -85,B 0,C 180,E1 -3815.085,E2 -3815.085} C_VEL
LIN {X 0,Y 537.992,Z 381.464,A -85,B 0,C 180,E1 -3817.878,E2 -3817.878} C_VEL
LIN {X 0,Y 538.051,Z 381.465,A -85,B 0,C 180,E1 -3820.776,E2 -3820.776} C_VEL
LIN {X 0,Y 538.013,Z 381.465,A -85,B 0,C 180,E1 -3824.072,E2 -3824.072} C_VEL
LIN {X 0,Y 538.001,Z 381.467,A -85,B 0,C 180,E1 -3827.016,E2 -3827.016} C_VEL
LIN {X 0,Y 538.051,Z 381.46,A -85,B 0,C 180,E1 -3829.253,E2 -3829.253} C_VEL
LIN {X 0,Y 537.991,Z 381.464,A -85,B 0,C 180,E1 -3832.122,E2 -3832.122} C_VEL
LIN {X 0,Y 537.997,Z 381.467,A -85,B 0,C 180,E1 -3834.915,E2 -3834.915} C_VEL
LIN {X 0,Y 538.021,Z 381.461,A -85,B 0,C 180,E1 -3837.617,E2 -3837.617} C_VEL
LIN {X 0,Y 538.014,Z 381.467,A -85,B 0,C 180,E1 -3840.239,E2 -3840.239} C_VEL
LIN {X 0,Y 538.075,Z 381.641,A -85,B 0,C 180,E1 -3842.428,E2 -3842.428} C_VEL
LIN {X 0,Y 540.295,Z 392.269,A -85,B 0,C 180,E1 -3843.836,E2 -3843.836} C_VEL
LIN {X 0,Y 539.881,Z 417.027,A -85,B 0,C 180,E1 -3846.81,E2 -3846.81} C_VEL
LIN {X 0,Y 539.414,Z 442.528,A -85,B 0,C 180,E1 -3849.851,E2 -3849.851} C_VEL
LIN {X 0,Y 538.925,Z 470.181,A -85,B 0,C 180,E1 -3853.133,E2 -3853.133} C_VEL
LIN {X 0,Y 538.664,Z 488.219,A -85,B 0,C 180,E1 -3855.259,E2 -3855.259} C_VEL
LIN {X 0,Y 539.674,Z 496.509,A -85,B 0,C 180,E1 -3855.42,E2 -3855.42} C_VEL
LIN {X 0,Y 539.335,Z 598.04,A -85,B 0,C 180,E1 -3856.794,E2 -3856.794} C_VEL
LIN {X 0,Y 539.191,Z 609.544,A -85,B 0,C 180,E1 -3857.078,E2 -3857.078} C_VEL
LIN {X 0,Y 538.996,Z 619.831,A -85,B 0,C 180,E1 -3857.433,E2 -3857.433} C_VEL
LIN {X 0,Y 538.879,Z 629.348,A -85,B 0,C 180,E1 -3857.86,E2 -3857.86} C_VEL
LIN {X 0,Y 538.701,Z 638.099,A -85,B 0,C 180,E1 -3858.343,E2 -3858.343} C_VEL
LIN {X 0,Y 538.555,Z 646.514,A -85,B 0,C 180,E1 -3858.902,E2 -3858.902} C_VEL
LIN {X 0,Y 538.328,Z 654.887,A -85,B 0,C 180,E1 -3859.564,E2 -3859.564} C_VEL
LIN {X 0,Y 538.16,Z 662.041,A -85,B 0,C 180,E1 -3860.226,E2 -3860.226} C_VEL
LIN {X 0,Y 537.98,Z 670.543,A -85,B 0,C 180,E1 -3861.17,E2 -3861.17} C_VEL
LIN {X 0,Y 537.83,Z 677.611,A -85,B 0,C 180,E1 -3862.114,E2 -3862.114} C_VEL
LIN {X 0,Y 537.74,Z 683.506,A -85,B 0,C 180,E1 -3863.056,E2 -3863.056} C_VEL
LIN {X 0,Y 537.696,Z 688.408,A -85,B 0,C 180,E1 -3863.998,E2 -3863.998} C_VEL
LIN {X 0,Y 537.54,Z 693.141,A -85,B 0,C 180,E1 -3865.125,E2 -3865.125} C_VEL
LIN {X 0,Y 537.591,Z 696.775,A -85,B 0,C 180,E1 -3866.252,E2 -3866.252} C_VEL
LIN {X 0,Y 537.551,Z 698.662,A -85,B 0,C 180,E1 -3867.002,E2 -3867.002} C_VEL
LIN {X 0,Y 537.49,Z 700.14,A -85,B 0,C 180,E1 -3867.752,E2 -3867.752} C_VEL
LIN {X 0,Y 537.442,Z 701.723,A -85,B 0,C 180,E1 -3869.251,E2 -3869.251} C_VEL
LIN {X 0,Y 537.442,Z 701.996,A -85,B 0,C 180,E1 -3870,E2 -3870} C_VEL
LIN {X 0,Y 537.452,Z 701.198,A -85,B 0,C 180,E1 -3871.499,E2 -3871.499} C_VEL
LIN {X 0,Y 537.49,Z 700.284,A -85,B 0,C 180,E1 -3872.248,E2 -3872.248} C_VEL
LIN {X 0,Y 537.591,Z 697.028,A -85,B 0,C 180,E1 -3873.748,E2 -3873.748} C_VEL
LIN {X 0,Y 537.54,Z 693.473,A -85,B 0,C 180,E1 -3874.875,E2 -3874.875} C_VEL
LIN {X 0,Y 537.667,Z 688.823,A -85,B 0,C 180,E1 -3876.003,E2 -3876.003} C_VEL
LIN {X 0,Y 537.698,Z 684.011,A -85,B 0,C 180,E1 -3876.944,E2 -3876.944} C_VEL
LIN {X 0,Y 537.817,Z 678.215,A -85,B 0,C 180,E1 -3877.887,E2 -3877.887} C_VEL
LIN {X 0,Y 537.94,Z 671.259,A -85,B 0,C 180,E1 -3878.831,E2 -3878.831} C_VEL
LIN {X 0,Y 538.111,Z 664.672,A -85,B 0,C 180,E1 -3879.586,E2 -3879.586} C_VEL
LIN {X 0,Y 538.257,Z 656.941,A -85,B 0,C 180,E1 -3880.343,E2 -3880.343} C_VEL
LIN {X 0,Y 538.489,Z 648.955,A -85,B 0,C 180,E1 -3881.004,E2 -3881.004} C_VEL
LIN {X 0,Y 538.652,Z 640.046,A -85,B 0,C 180,E1 -3881.625,E2 -3881.625} C_VEL
LIN {X 0,Y 538.824,Z 631.088,A -85,B 0,C 180,E1 -3882.141,E2 -3882.141} C_VEL
LIN {X 0,Y 538.989,Z 622.025,A -85,B 0,C 180,E1 -3882.568,E2 -3882.568} C_VEL
LIN {X 0,Y 539.158,Z 611.677,A -85,B 0,C 180,E1 -3882.947,E2 -3882.947} C_VEL
LIN {X 0,Y 539.344,Z 600.17,A -85,B 0,C 180,E1 -3883.254,E2 -3883.254} C_VEL
LIN {X 0,Y 539.453,Z 575.753,A -85,B 0,C 180,E1 -3883.611,E2 -3883.611} C_VEL
LIN {X 0,Y 539.564,Z 495,A -85,B 0,C 180,E1 -3884.693,E2 -3884.693} C_VEL
LIN {X 0,Y 538.655,Z 488.029,A -85,B 0,C 180,E1 -3884.84,E2 -3884.84} C_VEL
LIN {X 0,Y 539.021,Z 462.583,A -85,B 0,C 180,E1 -3887.859,E2 -3887.859} C_VEL
LIN {X 0,Y 539.483,Z 437.899,A -85,B 0,C 180,E1 -3890.793,E2 -3890.793} C_VEL
LIN {X 0,Y 539.904,Z 416.153,A -85,B 0,C 180,E1 -3893.392,E2 -3893.392} C_VEL
LIN {X 0,Y 540.278,Z 392.393,A -85,B 0,C 180,E1 -3896.249,E2 -3896.249} C_VEL
LIN {X 0,Y 538.049,Z 381.598,A -85,B 0,C 180,E1 -3897.676,E2 -3897.676} C_VEL
LIN {X 0,Y 538.01,Z 381.466,A -85,B 0,C 180,E1 -3900.628,E2 -3900.628} C_VEL
LIN {X 0,Y 538.05,Z 381.465,A -85,B 0,C 180,E1 -3903.283,E2 -3903.283} C_VEL
LIN {X 0,Y 537.965,Z 381.471,A -85,B 0,C 180,E1 -3906.007,E2 -3906.007} C_VEL
LIN {X 0,Y 538.012,Z 381.465,A -85,B 0,C 180,E1 -3908.831,E2 -3908.831} C_VEL
LIN {X 0,Y 537.987,Z 381.473,A -85,B 0,C 180,E1 -3911.873,E2 -3911.873} C_VEL
LIN {X 0,Y 537.996,Z 381.459,A -85,B 0,C 180,E1 -3914.864,E2 -3914.864} C_VEL
LIN {X 0,Y 537.99,Z 381.469,A -85,B 0,C 180,E1 -3917.211,E2 -3917.211} C_VEL
LIN {X 0,Y 538.013,Z 381.464,A -85,B 0,C 180,E1 -3920.418,E2 -3920.418} C_VEL
LIN {X 0,Y 537.994,Z 381.464,A -85,B 0,C 180,E1 -3923.064,E2 -3923.064} C_VEL
LIN {X 0,Y 538.001,Z 381.468,A -85,B 0,C 180,E1 -3925.825,E2 -3925.825} C_VEL
LIN {X 0,Y 538.012,Z 381.464,A -85,B 0,C 180,E1 -3928.499,E2 -3928.499} C_VEL
LIN {X 0,Y 537.988,Z 381.465,A -85,B 0,C 180,E1 -3931.095,E2 -3931.095} C_VEL
LIN {X 0,Y 537.985,Z 381.475,A -85,B 0,C 180,E1 -3933.63,E2 -3933.63} C_VEL
LIN {X 0,Y 538.011,Z 381.463,A -85,B 0,C 180,E1 -3936.122,E2 -3936.122} C_VEL
LIN {X 0,Y 538.019,Z 381.462,A -85,B 0,C 180,E1 -3938.546,E2 -3938.546} C_VEL
LIN {X 0,Y 538.011,Z 381.462,A -85,B 0,C 180,E1 -3940.939,E2 -3940.939} C_VEL
LIN {X 0,Y 537.975,Z 381.467,A -85,B 0,C 180,E1 -3943.297,E2 -3943.297} C_VEL
LIN {X 0,Y 538.055,Z 381.465,A -85,B 0,C 180,E1 -3945.63,E2 -3945.63} C_VEL
LIN {X 0,Y 538.027,Z 381.455,A -85,B 0,C 180,E1 -3948.7,E2 -3948.7} C_VEL
LIN {X 0,Y 538.043,Z 381.468,A -85,B 0,C 180,E1 -3951.739,E2 -3951.739} C_VEL
LIN {X 0,Y 538.126,Z 381.444,A -85,B 0,C 180,E1 -3954.755,E2 -3954.755} C_VEL
LIN {X 0,Y 538.164,Z 381.451,A -85,B 0,C 180,E1 -3957.755,E2 -3957.755} C_VEL
LIN {X 0,Y 538.163,Z 381.448,A -85,B 0,C 180,E1 -3960,E2 -3960} C_VEL
LIN {X 0,Y 538.114,Z 381.444,A -85,B 0,C 180,E1 -3962.995,E2 -3962.995} C_VEL
LIN {X 0,Y 538.083,Z 381.46,A -85,B 0,C 180,E1 -3965.998,E2 -3965.998} C_VEL
LIN {X 0,Y 538.029,Z 381.457,A -85,B 0,C 180,E1 -3969.018,E2 -3969.018} C_VEL
LIN {X 0,Y 538.041,Z 381.464,A -85,B 0,C 180,E1 -3972.063,E2 -3972.063} C_VEL
LIN {X 0,Y 537.99,Z 381.465,A -85,B 0,C 180,E1 -3975.145,E2 -3975.145} C_VEL
LIN {X 0,Y 537.986,Z 381.468,A -85,B 0,C 180,E1 -3978.272,E2 -3978.272} C_VEL
LIN {X 0,Y 537.978,Z 381.467,A -85,B 0,C 180,E1 -3980.654,E2 -3980.654} C_VEL
LIN {X 0,Y 538.009,Z 381.459,A -85,B 0,C 180,E1 -3983.072,E2 -3983.072} C_VEL
LIN {X 0,Y 537.986,Z 381.472,A -85,B 0,C 180,E1 -3985.658,E2 -3985.658} C_VEL
LIN {X 0,Y 537.973,Z 381.469,A -85,B 0,C 180,E1 -3988.054,E2 -3988.054} C_VEL
LIN {X 0,Y 538.005,Z 381.463,A -85,B 0,C 180,E1 -3990.628,E2 -3990.628} C_VEL
LIN {X 0,Y 538.023,Z 381.463,A -85,B 0,C 180,E1 -3993.278,E2 -3993.278} C_VEL
LIN {X 0,Y 537.957,Z 381.477,A -85,B 0,C 180,E1 -3996.008,E2 -3996.008} C_VEL
LIN {X 0,Y 537.986,Z 381.463,A -85,B 0,C 180,E1 -3998.833,E2 -3998.833} C_VEL
LIN {X 0,Y 537.976,Z 381.462,A -85,B 0,C 180,E1 -4001.872,E2 -4001.872} C_VEL
LIN {X 0,Y 537.991,Z 381.465,A -85,B 0,C 180,E1 -4004.864,E2 -4004.864} C_VEL
LIN {X 0,Y 537.972,Z 381.467,A -85,B 0,C 180,E1 -4007.209,E2 -4007.209} C_VEL
LIN {X 0,Y 537.979,Z 381.468,A -85,B 0,C 180,E1 -4010.422,E2 -4010.422} C_VEL
LIN {X 0,Y 537.953,Z 381.471,A -85,B 0,C 180,E1 -4013.061,E2 -4013.061} C_VEL
LIN {X 0,Y 537.991,Z 381.475,A -85,B 0,C 180,E1 -4015.824,E2 -4015.824} C_VEL
LIN {X 0,Y 537.991,Z 381.471,A -85,B 0,C 180,E1 -4018.497,E2 -4018.497} C_VEL
LIN {X 0,Y 538.018,Z 381.601,A -85,B 0,C 180,E1 -4021.723,E2 -4021.723} C_VEL
LIN {X 0,Y 540.397,Z 392.158,A -85,B 0,C 180,E1 -4023.132,E2 -4023.132} C_VEL
LIN {X 0,Y 540.153,Z 411.353,A -85,B 0,C 180,E1 -4025.395,E2 -4025.395} C_VEL
LIN {X 0,Y 539.627,Z 435.523,A -85,B 0,C 180,E1 -4028.211,E2 -4028.211} C_VEL
LIN {X 0,Y 539.246,Z 458.032,A -85,B 0,C 180,E1 -4030.787,E2 -4030.787} C_VEL
LIN {X 0,Y 538.799,Z 484.055,A -85,B 0,C 180,E1 -4033.713,E2 -4033.713} C_VEL
LIN {X 0,Y 538.653,Z 497.584,A -85,B 0,C 180,E1 -4035.212,E2 -4035.212} C_VEL
LIN {X 0,Y 539.681,Z 505.773,A -85,B 0,C 180,E1 -4035.371,E2 -4035.371} C_VEL
LIN {X 0,Y 539.335,Z 607.937,A -85,B 0,C 180,E1 -4036.746,E2 -4036.746} C_VEL
LIN {X 0,Y 539.173,Z 620.448,A -85,B 0,C 180,E1 -4037.054,E2 -4037.054} C_VEL
LIN {X 0,Y 538.97,Z 633.364,A -85,B 0,C 180,E1 -4037.527,E2 -4037.527} C_VEL
LIN {X 0,Y 538.788,Z 644.786,A -85,B 0,C 180,E1 -4038.095,E2 -4038.095} C_VEL
LIN {X 0,Y 538.545,Z 655.899,A -85,B 0,C 180,E1 -4038.807,E2 -4038.807} C_VEL
LIN {X 0,Y 538.269,Z 666.534,A -85,B 0,C 180,E1 -4039.657,E2 -4039.657} C_VEL
LIN {X 0,Y 538.068,Z 676.112,A -85,B 0,C 180,E1 -4040.603,E2 -4040.603} C_VEL
LIN {X 0,Y 537.921,Z 683.959,A -85,B 0,C 180,E1 -4041.548,E2 -4041.548} C_VEL
LIN {X 0,Y 537.755,Z 691.621,A -85,B 0,C 180,E1 -4042.679,E2 -4042.679} C_VEL
LIN {X 0,Y 537.693,Z 698.679,A -85,B 0,C 180,E1 -4043.998,E2 -4043.998} C_VEL
LIN {X 0,Y 537.54,Z 703.372,A -85,B 0,C 180,E1 -4045.125,E2 -4045.125} C_VEL
LIN {X 0,Y 537.591,Z 706.958,A -85,B 0,C 180,E1 -4046.252,E2 -4046.252} C_VEL
LIN {X 0,Y 537.551,Z 708.807,A -85,B 0,C 180,E1 -4047.002,E2 -4047.002} C_VEL
LIN {X 0,Y 537.451,Z 711.182,A -85,B 0,C 180,E1 -4048.501,E2 -4048.501} C_VEL
LIN {X 0,Y 537.442,Z 712,A -85,B 0,C 180,E1 -4050,E2 -4050} C_VEL
LIN {X 0,Y 537.451,Z 711.184,A -85,B 0,C 180,E1 -4051.499,E2 -4051.499} C_VEL
LIN {X 0,Y 537.551,Z 708.81,A -85,B 0,C 180,E1 -4052.998,E2 -4052.998} C_VEL
LIN {X 0,Y 537.603,Z 705.895,A -85,B 0,C 180,E1 -4054.123,E2 -4054.123} C_VEL
LIN {X 0,Y 537.587,Z 701.948,A -85,B 0,C 180,E1 -4055.251,E2 -4055.251} C_VEL
LIN {X 0,Y 537.65,Z 697.08,A -85,B 0,C 180,E1 -4056.335,E2 -4056.335} C_VEL
LIN {X 0,Y 537.791,Z 690.467,A -85,B 0,C 180,E1 -4057.509,E2 -4057.509} C_VEL
LIN {X 0,Y 537.972,Z 682.477,A -85,B 0,C 180,E1 -4058.64,E2 -4058.64} C_VEL
LIN {X 0,Y 538.145,Z 674.333,A -85,B 0,C 180,E1 -4059.585,E2 -4059.585} C_VEL
LIN {X 0,Y 538.364,Z 664.397,A -85,B 0,C 180,E1 -4060.531,E2 -4060.531} C_VEL
LIN {X 0,Y 538.579,Z 654.592,A -85,B 0,C 180,E1 -4061.288,E2 -4061.288} C_VEL
LIN {X 0,Y 538.805,Z 643.695,A -85,B 0,C 180,E1 -4061.964,E2 -4061.964} C_VEL
LIN {X 0,Y 538.969,Z 631.101,A -85,B 0,C 180,E1 -4062.568,E2 -4062.568} C_VEL
LIN {X 0,Y 539.208,Z 618.087,A -85,B 0,C 180,E1 -4063.017,E2 -4063.017} C_VEL
LIN {X 0,Y 539.346,Z 605.104,A -85,B 0,C 180,E1 -4063.301,E2 -4063.301} C_VEL
LIN {X 0,Y 539.52,Z 504.389,A -85,B 0,C 180,E1 -4064.649,E2 -4064.649} C_VEL
LIN {X 0,Y 538.666,Z 497.502,A -85,B 0,C 180,E1 -4064.787,E2 -4064.787} C_VEL
LIN {X 0,Y 538.978,Z 469.599,A -85,B 0,C 180,E1 -4067.845,E2 -4067.845} C_VEL
LIN {X 0,Y 539.384,Z 442.979,A -85,B 0,C 180,E1 -4070.797,E2 -4070.797} C_VEL
LIN {X 0,Y 539.798,Z 415.117,A -85,B 0,C 180,E1 -4073.945,E2 -4073.945} C_VEL
LIN {X 0,Y 540.071,Z 393.185,A -85,B 0,C 180,E1 -4076.468,E2 -4076.468} C_VEL
LIN {X 0,Y 539.284,Z 387.738,A -85,B 0,C 180,E1 -4077.137,E2 -4077.137} C_VEL
LIN {X 0,Y 537.992,Z 381.575,A -85,B 0,C 180,E1 -4077.97,E2 -4077.97} C_VEL
LIN {X 0,Y 537.989,Z 381.471,A -85,B 0,C 180,E1 -4080.629,E2 -4080.629} C_VEL
LIN {X 0,Y 538,Z 381.468,A -85,B 0,C 180,E1 -4083.275,E2 -4083.275} C_VEL
LIN {X 0,Y 537.955,Z 381.479,A -85,B 0,C 180,E1 -4086.008,E2 -4086.008} C_VEL
LIN {X 0,Y 537.986,Z 381.468,A -85,B 0,C 180,E1 -4088.833,E2 -4088.833} C_VEL
LIN {X 0,Y 537.976,Z 381.476,A -85,B 0,C 180,E1 -4091.872,E2 -4091.872} C_VEL
LIN {X 0,Y 537.995,Z 381.466,A -85,B 0,C 180,E1 -4094.864,E2 -4094.864} C_VEL
LIN {X 0,Y 537.975,Z 381.47,A -85,B 0,C 180,E1 -4097.209,E2 -4097.209} C_VEL
LIN {X 0,Y 538.012,Z 381.464,A -85,B 0,C 180,E1 -4100.418,E2 -4100.418} C_VEL
LIN {X 0,Y 537.993,Z 381.468,A -85,B 0,C 180,E1 -4103.064,E2 -4103.064} C_VEL
LIN {X 0,Y 538.014,Z 381.469,A -85,B 0,C 180,E1 -4105.826,E2 -4105.826} C_VEL
LIN {X 0,Y 538.011,Z 381.464,A -85,B 0,C 180,E1 -4108.499,E2 -4108.499} C_VEL
LIN {X 0,Y 538.021,Z 381.467,A -85,B 0,C 180,E1 -4111.097,E2 -4111.097} C_VEL
LIN {X 0,Y 538.016,Z 381.469,A -85,B 0,C 180,E1 -4113.632,E2 -4113.632} C_VEL
LIN {X 0,Y 538.01,Z 381.466,A -85,B 0,C 180,E1 -4116.122,E2 -4116.122} C_VEL
LIN {X 0,Y 538.041,Z 381.468,A -85,B 0,C 180,E1 -4119.349,E2 -4119.349} C_VEL
LIN {X 0,Y 538.039,Z 381.463,A -85,B 0,C 180,E1 -4122.468,E2 -4122.468} C_VEL
LIN {X 0,Y 538.134,Z 381.613,A -85,B 0,C 180,E1 -4125.602,E2 -4125.602} C_VEL
LIN {X 0,Y 538.354,Z 382.725,A -85,B 0,C 180,E1 -4125.73,E2 -4125.73} C_VEL
LIN {X 0,Y 539.613,Z 386.729,A -85,B 0,C 180,E1 -4125.829,E2 -4125.829} C_VEL
LIN {X 0,Y 539.246,Z 462.272,A -85,B 0,C 180,E1 -4126.888,E2 -4126.888} C_VEL
LIN {X 0,Y 539.196,Z 476.081,A -85,B 0,C 180,E1 -4127.246,E2 -4127.246} C_VEL
LIN {X 0,Y 539.043,Z 488.397,A -85,B 0,C 180,E1 -4127.72,E2 -4127.72} C_VEL
LIN {X 0,Y 538.86,Z 499.781,A -85,B 0,C 180,E1 -4128.314,E2 -4128.314} C_VEL
LIN {X 0,Y 538.689,Z 510.16,A -85,B 0,C 180,E1 -4129,E2 -4129} C_VEL
LIN {X 0,Y 538.463,Z 520.515,A -85,B 0,C 180,E1 -4129.851,E2 -4129.851} C_VEL
LIN {X 0,Y 538.281,Z 529.801,A -85,B 0,C 180,E1 -4130.797,E2 -4130.797} C_VEL
LIN {X 0,Y 538.098,Z 538.684,A -85,B 0,C 180,E1 -4131.929,E2 -4131.929} C_VEL
LIN {X 0,Y 537.97,Z 544.938,A -85,B 0,C 180,E1 -4132.909,E2 -4132.909} C_VEL
LIN {X 0,Y 537.903,Z 550.6,A -85,B 0,C 180,E1 -4134,E2 -4134} C_VEL
LIN {X 0,Y 537.747,Z 555.26,A -85,B 0,C 180,E1 -4135.127,E2 -4135.127} C_VEL
LIN {X 0,Y 537.72,Z 558.856,A -85,B 0,C 180,E1 -4136.253,E2 -4136.253} C_VEL
LIN {X 0,Y 537.618,Z 562.073,A -85,B 0,C 180,E1 -4137.752,E2 -4137.752} C_VEL
LIN {X 0,Y 537.601,Z 563.614,A -85,B 0,C 180,E1 -4139.251,E2 -4139.251} C_VEL
LIN {X 0,Y 537.595,Z 563.853,A -85,B 0,C 180,E1 -4140,E2 -4140} C_VEL
LIN {X 0,Y 537.598,Z 563.055,A -85,B 0,C 180,E1 -4141.498,E2 -4141.498} C_VEL
LIN {X 0,Y 537.613,Z 562.119,A -85,B 0,C 180,E1 -4142.248,E2 -4142.248} C_VEL
LIN {X 0,Y 537.669,Z 560.745,A -85,B 0,C 180,E1 -4142.997,E2 -4142.997} C_VEL
LIN {X 0,Y 537.731,Z 556.723,A -85,B 0,C 180,E1 -4144.498,E2 -4144.498} C_VEL
LIN {X 0,Y 537.809,Z 552.49,A -85,B 0,C 180,E1 -4145.625,E2 -4145.625} C_VEL
LIN {X 0,Y 537.862,Z 547.079,A -85,B 0,C 180,E1 -4146.754,E2 -4146.754} C_VEL
LIN {X 0,Y 537.998,Z 540.26,A -85,B 0,C 180,E1 -4147.884,E2 -4147.884} C_VEL
LIN {X 0,Y 538.191,Z 533.312,A -85,B 0,C 180,E1 -4148.826,E2 -4148.826} C_VEL
LIN {X 0,Y 538.327,Z 524.913,A -85,B 0,C 180,E1 -4149.772,E2 -4149.772} C_VEL
LIN {X 0,Y 538.574,Z 515.712,A -85,B 0,C 180,E1 -4150.622,E2 -4150.622} C_VEL
LIN {X 0,Y 538.816,Z 505.051,A -85,B 0,C 180,E1 -4151.419,E2 -4151.419} C_VEL
LIN {X 0,Y 538.96,Z 492.82,A -85,B 0,C 180,E1 -4152.138,E2 -4152.138} C_VEL
LIN {X 0,Y 539.1,Z 480.993,A -85,B 0,C 180,E1 -4152.661,E2 -4152.661} C_VEL
LIN {X 0,Y 539.252,Z 469.197,A -85,B 0,C 180,E1 -4153.04,E2 -4153.04} C_VEL
